KUKA KRL program: MyProgram_094().src

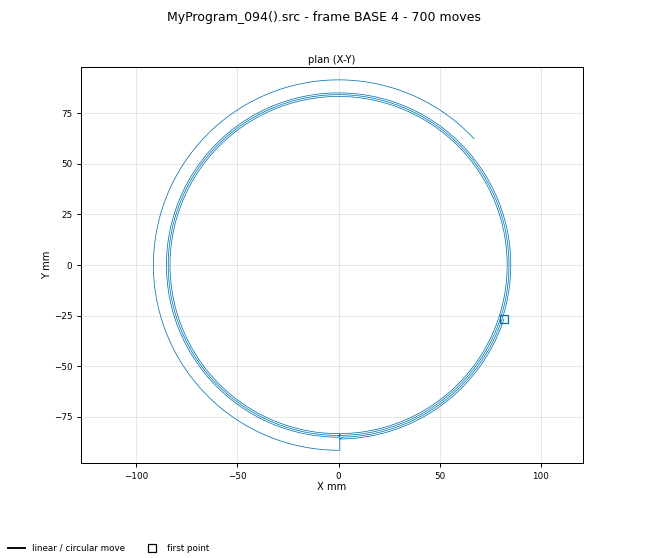
[picture p0: tool path of MyProgram_094().src in frame BASE 4, 700 of 700 moves have a stored position in this frame; points joined in program order, loops and branches not executed]
&ACCESS RVP
&REL 1
&PARAM TEMPLATE = C:\KRC\Roboter\Template\vorgabe
&PARAM EDITMASK = *
DEF MyProgram_094()
; ---- Setting reference (Base) ----
$BASE = BASE_DATA[4]

; --------------------------
; ---- Setting tool (TCP) ----
$TOOL = TOOL_DATA[3]
; --------------------------

$VEL.CP = VEL_APROX_PRINT
Startdeposition()
$VEL.CP = VEL_PRINT
LIN {X 81.733,Y -26.6851,Z 88,A -23.6392,B 24.9182,C -2.0882,E1 25.1514,E2 468.5643} C_DIS
LIN {X 80.2475,Y -30.8683,Z 88,A -26.5648,B 24.9188,C -2.0802,E1 25.1486,E2 471.4924} C_DIS
LIN {X 77.8159,Y -36.5664,Z 88,A -30.6029,B 24.9196,C -2.0708,E1 25.1441,E2 475.5307} C_DIS
LIN {X 76.3718,Y -39.4947,Z 88,A -32.5846,B 24.9196,C -2.071,E1 25.1416,E2 477.5014} C_DIS
LIN {X 74.1282,Y -43.5589,Z 88,A -35.9674,B 24.921,C -2.0522,E1 25.1369,E2 480.911} C_DIS
LIN {X 71.5565,Y -47.6671,Z 88,A -38.965,B 24.9211,C -2.051,E1 25.1324,E2 483.8964} C_DIS
LIN {X 70.1934,Y -49.6508,Z 88,A -41.3471,B 24.9235,C -2.0204,E1 25.1285,E2 486.3392} C_DIS
LIN {X 67.8657,Y -52.7894,Z 88,A -43.5721,B 24.923,C -2.0261,E1 25.1247,E2 488.5401} C_DIS
LIN {X 64.4289,Y -56.934,Z 88,A -46.6091,B 24.9223,C -2.0354,E1 25.1193,E2 491.5414} C_DIS
LIN {X 62.1331,Y -59.4299,Z 88,A -49.1933,B 24.9236,C -2.0188,E1 25.1144,E2 494.1534} C_DIS
LIN {X 59.2198,Y -62.3328,Z 88,A -52.3338,B 24.9251,C -1.999,E1 25.108,E2 497.3276} C_DIS
LIN {X 56.7113,Y -64.6234,Z 88,A -53.6632,B 24.9231,C -2.0249,E1 25.1054,E2 498.5904} C_DIS
LIN {X 54.5742,Y -66.438,Z 88,A -56.1783,B 24.9251,C -1.9992,E1 25.0998,E2 501.1567} C_DIS
LIN {X 49.6783,Y -70.1747,Z 88,A -60.1672,B 24.9254,C -1.9944,E1 25.0909,E2 505.1426} C_DIS
LIN {X 47.2805,Y -71.8114,Z 88,A -62.4831,B 24.9266,C -1.9781,E1 25.0854,E2 507.4893} C_DIS
LIN {X 44.2965,Y -73.6906,Z 88,A -64.087,B 24.9251,C -1.9982,E1 25.0817,E2 509.0406} C_DIS
LIN {X 41.297,Y -75.4121,Z 88,A -66.6065,B 24.926,C -1.9871,E1 25.0756,E2 511.5791} C_DIS
LIN {X 38.2378,Y -77.0077,Z 88,A -68.7734,B 24.926,C -1.9876,E1 25.0702,E2 513.7388} C_DIS
LIN {X 34.3008,Y -78.8402,Z 88,A -72.2408,B 24.9276,C -1.9646,E1 25.0612,E2 517.2521} C_DIS
LIN {X 31.2368,Y -80.1038,Z 88,A -73.7753,B 24.9262,C -1.9833,E1 25.0574,E2 518.7388} C_DIS
LIN {X 28.0288,Y -81.2822,Z 88,A -76.7376,B 24.9281,C -1.9583,E1 25.0494,E2 521.7543} C_DIS
LIN {X 24.8043,Y -82.3237,Z 88,A -78.4493,B 24.927,C -1.9732,E1 25.045,E2 523.4276} C_DIS
LIN {X 21.2594,Y -83.3089,Z 88,A -81.7956,B 24.9293,C -1.9422,E1 25.0358,E2 526.8422} C_DIS
LIN {X 16.7926,Y -84.3241,Z 88,A -83.7415,B 24.9269,C -1.9746,E1 25.0307,E2 528.7088} C_DIS
LIN {X 10.7108,Y -85.3095,Z 88,A -87.865,B 24.9272,C -1.9711,E1 25.0193,E2 532.8369} C_DIS
LIN {X 7.4694,Y -85.6546,Z 88,A -90.1854,B 24.9276,C -1.9652,E1 25.0128,E2 535.1697} C_DIS
LIN {X 4.6796,Y -85.8512,Z 88,A -92.9626,B 24.9297,C -1.9359,E1 25.0049,E2 538.0153} C_DIS
LIN {X 0.5582,Y -85.9679,Z 88,A -93.1523,B 24.9238,C -2.0159,E1 25.0049,E2 538.0153} C_DIS
Enddeposition()
LIN {X 0.5582,Y -85.9679,Z 88,A -93.1523,B 24.9238,C -2.0159,E1 25.0049,E2 538.0153} C_DIS
Startdeposition()
$VEL.CP = VEL_PRINT
LIN {X 1.674,Y -85.0811,Z 88,A -92.9521,B 24.924,C -2.0134,E1 25.0054,E2 537.8212} C_DIS
LIN {X 5.5624,Y -84.9157,Z 88,A -89.8499,B 24.9227,C -2.0298,E1 25.0141,E2 534.6812} C_DIS
LIN {X 9.1586,Y -84.6037,Z 88,A -87.9756,B 24.924,C -2.0134,E1 25.0192,E2 532.8471} C_DIS
LIN {X 12.5486,Y -84.1684,Z 88,A -85.0762,B 24.9224,C -2.0342,E1 25.0274,E2 529.901} C_DIS
LIN {X 16.1894,Y -83.5434,Z 88,A -83.3504,B 24.9241,C -2.0116,E1 25.032,E2 528.2306} C_DIS
LIN {X 20.7796,Y -82.5225,Z 88,A -80.0885,B 24.9237,C -2.0177,E1 25.0409,E2 524.9588} C_DIS
LIN {X 23.9194,Y -81.6672,Z 88,A -77.9107,B 24.9235,C -2.0197,E1 25.0467,E2 522.78} C_DIS
LIN {X 26.4302,Y -80.8894,Z 88,A -75.3855,B 24.9215,C -2.0465,E1 25.0536,E2 520.1959} C_DIS
LIN {X 30.2485,Y -79.5401,Z 88,A -73.5932,B 24.9235,C -2.0195,E1 25.0581,E2 518.4715} C_DIS
LIN {X 33.1948,Y -78.3563,Z 88,A -71.1205,B 24.9225,C -2.0335,E1 25.0645,E2 515.9712} C_DIS
LIN {X 36.3155,Y -76.9608,Z 88,A -68.9238,B 24.9225,C -2.0336,E1 25.0701,E2 513.7799} C_DIS
LIN {X 39.5256,Y -75.3613,Z 88,A -66.5837,B 24.9223,C -2.0352,E1 25.0759,E2 511.4426} C_DIS
LIN {X 42.557,Y -73.692,Z 88,A -64.2486,B 24.922,C -2.0395,E1 25.0816,E2 509.1042} C_DIS
LIN {X 47.2525,Y -70.7745,Z 88,A -60.7688,B 24.922,C -2.0385,E1 25.0898,E2 505.638} C_DIS
LIN {X 50.0783,Y -68.8026,Z 88,A -58.0174,B 24.9206,C -2.0576,E1 25.0961,E2 502.8509} C_DIS
LIN {X 53.2996,Y -66.3382,Z 88,A -55.444,B 24.9206,C -2.0582,E1 25.1017,E2 500.2856} C_DIS
LIN {X 56.1485,Y -63.9452,Z 88,A -52.9116,B 24.9201,C -2.0648,E1 25.1071,E2 497.7476} C_DIS
LIN {X 58.92,Y -61.4008,Z 88,A -50.5533,B 24.9201,C -2.0648,E1 25.1119,E2 495.3988} C_DIS
LIN {X 61.2054,Y -59.1226,Z 88,A -48.345,B 24.9195,C -2.0714,E1 25.1162,E2 493.1845} C_DIS
LIN {X 63.807,Y -56.3066,Z 88,A -45.7587,B 24.919,C -2.078,E1 25.1211,E2 490.594} C_DIS
LIN {X 66.1479,Y -53.5354,Z 88,A -43.3524,B 24.9186,C -2.0832,E1 25.1254,E2 488.1866} C_DIS
LIN {X 68.597,Y -50.3592,Z 88,A -40.3906,B 24.9173,C -2.0994,E1 25.1304,E2 485.2007} C_DIS
LIN {X 70.5872,Y -47.5297,Z 88,A -37.8925,B 24.9164,C -2.1116,E1 25.1343,E2 482.6861} C_DIS
LIN {X 73.7566,Y -42.4447,Z 88,A -34.5122,B 24.9172,C -2.1007,E1 25.1391,E2 479.3487} C_DIS
LIN {X 74.9881,Y -40.2309,Z 88,A -32.7904,B 24.9168,C -2.1062,E1 25.1414,E2 477.623} C_DIS
LIN {X 76.4162,Y -37.4472,Z 88,A -30.7153,B 24.9164,C -2.1114,E1 25.1441,E2 475.5467} C_DIS
LIN {X 77.6659,Y -34.7797,Z 88,A -28.1064,B 24.9142,C -2.1389,E1 25.1471,E2 472.8871} C_DIS
LIN {X 78.9315,Y -31.804,Z 88,A -26.5631,B 24.9154,C -2.1236,E1 25.1487,E2 471.3883} C_DIS
LIN {X 80.7731,Y -26.7857,Z 88,A -22.8946,B 24.9143,C -2.1371,E1 25.1522,E2 467.7086} C_DIS
LIN {X 81.7527,Y -23.6278,Z 88,A -20.5927,B 24.9136,C -2.1466,E1 25.154,E2 465.3972} C_DIS
LIN {X 82.5245,Y -20.7718,Z 88,A -18.9002,B 24.9139,C -2.1426,E1 25.1552,E2 463.724} C_DIS
LIN {X 83.2588,Y -17.6004,Z 88,A -16.4666,B 24.9127,C -2.1579,E1 25.1567,E2 461.2684} C_DIS
LIN {X 84.1496,Y -12.6706,Z 88,A -13.1028,B 24.9118,C -2.1683,E1 25.1583,E2 457.8998} C_DIS
LIN {X 84.5645,Y -9.5168,Z 88,A -11.0727,B 24.9116,C -2.1713,E1 25.1589,E2 455.8746} C_DIS
LIN {X 84.7904,Y -7.2374,Z 88,A -9.3098,B 24.9105,C -2.1839,E1 25.1594,E2 454.0925} C_DIS
LIN {X 85.0939,Y -0.8863,Z 88,A -4.8253,B 24.9088,C -2.2046,E1 25.1598,E2 449.5858} C_DIS
LIN {X 85.0004,Y 4.0858,Z 88,A -1.7552,B 24.9088,C -2.2056,E1 25.1595,E2 446.5315} C_DIS
LIN {X 84.6266,Y 8.9405,Z 88,A 0.8808,B 24.9097,C -2.194,E1 25.1589,E2 443.9385} C_DIS
LIN {X 84.3639,Y 11.1521,Z 88,A 3.4937,B 24.9061,C -2.237,E1 25.1579,E2 441.2396} C_DIS
LIN {X 83.7907,Y 14.8575,Z 88,A 5.1462,B 24.908,C -2.2148,E1 25.1572,E2 439.6491} C_DIS
LIN {X 83.0057,Y 18.7565,Z 88,A 8.0759,B 24.9066,C -2.2317,E1 25.1555,E2 436.6967} C_DIS
LIN {X 82.2132,Y 21.9689,Z 88,A 10.2169,B 24.9063,C -2.2355,E1 25.154,E2 434.559} C_DIS
LIN {X 81.1968,Y 25.4703,Z 88,A 12.5277,B 24.906,C -2.238,E1 25.1521,E2 432.2556} C_DIS
LIN {X 80.3027,Y 28.1614,Z 88,A 14.4713,B 24.9055,C -2.2448,E1 25.1504,E2 430.3068} C_DIS
LIN {X 79.2539,Y 30.9907,Z 88,A 16.5091,B 24.905,C -2.2509,E1 25.1483,E2 428.2659} C_DIS
LIN {X 78.0763,Y 33.8481,Z 88,A 18.5822,B 24.9045,C -2.2566,E1 25.1461,E2 426.1907} C_DIS
LIN {X 76.2957,Y 37.6904,Z 88,A 21.4623,B 24.9037,C -2.2656,E1 25.1426,E2 423.3051} C_DIS
LIN {X 75.2676,Y 39.7036,Z 88,A 23.177,B 24.9028,C -2.2762,E1 25.1404,E2 421.5741} C_DIS
LIN {X 73.4534,Y 42.9689,Z 88,A 25.4627,B 24.9028,C -2.2752,E1 25.1372,E2 419.3027} C_DIS
LIN {X 71.9394,Y 45.4587,Z 88,A 27.564,B 24.902,C -2.285,E1 25.1341,E2 417.1889} C_DIS
LIN {X 69.9909,Y 48.4035,Z 88,A 29.4184,B 24.903,C -2.2735,E1 25.1313,E2 415.3709} C_DIS
LIN {X 68.6867,Y 50.2366,Z 88,A 31.7063,B 24.9005,C -2.3031,E1 25.1274,E2 413.024} C_DIS
LIN {X 65.9916,Y 53.7283,Z 88,A 34.3193,B 24.9009,C -2.2982,E1 25.1229,E2 410.4348} C_DIS
LIN {X 63.8485,Y 56.2591,Z 88,A 36.2398,B 24.9014,C -2.2929,E1 25.1195,E2 408.5355} C_DIS
LIN {X 61.2216,Y 59.1058,Z 88,A 39.0377,B 24.9003,C -2.3049,E1 25.1141,E2 405.7215} C_DIS
LIN {X 58.927,Y 61.394,Z 88,A 41.2254,B 24.8999,C -2.3097,E1 25.1097,E2 403.5316} C_DIS
LIN {X 57.0263,Y 63.1642,Z 88,A 43.4545,B 24.8982,C -2.3291,E1 25.105,E2 401.2657} C_DIS
LIN {X 53.3912,Y 66.2648,Z 88,A 46.3212,B 24.8987,C -2.3236,E1 25.0989,E2 398.423} C_DIS
LIN {X 50.359,Y 68.5971,Z 88,A 48.6255,B 24.8991,C -2.3192,E1 25.0938,E2 396.1373} C_DIS
LIN {X 47.5261,Y 70.5897,Z 88,A 51.2112,B 24.898,C -2.3313,E1 25.0878,E2 393.5317} C_DIS
LIN {X 43.9489,Y 72.8708,Z 88,A 54.1354,B 24.8974,C -2.3378,E1 25.0809,E2 390.6014} C_DIS
LIN {X 40.6311,Y 74.771,Z 88,A 56.4193,B 24.898,C -2.332,E1 25.0754,E2 388.338} C_DIS
LIN {X 37.416,Y 76.4317,Z 88,A 58.942,B 24.8974,C -2.3378,E1 25.0691,E2 385.8084} C_DIS
LIN {X 33.4143,Y 78.2638,Z 88,A 62.1381,B 24.8965,C -2.3486,E1 25.0608,E2 382.5946} C_DIS
LIN {X 29.8776,Y 79.6805,Z 88,A 64.4126,B 24.8971,C -2.3418,E1 25.055,E2 380.3411} C_DIS
LIN {X 26.993,Y 80.7032,Z 88,A 66.5381,B 24.8968,C -2.3456,E1 25.0494,E2 378.2108} C_DIS
LIN {X 24.0987,Y 81.614,Z 88,A 68.2506,B 24.8975,C -2.3368,E1 25.0448,E2 376.5225} C_DIS
LIN {X 22.2097,Y 82.1481,Z 88,A 69.9297,B 24.8965,C -2.3489,E1 25.0403,E2 374.8174} C_DIS
LIN {X 18.6575,Y 83.0286,Z 88,A 72.4715,B 24.8961,C -2.3526,E1 25.0333,E2 372.2702} C_DIS
LIN {X 15.4369,Y 83.6865,Z 88,A 74.8346,B 24.8957,C -2.3582,E1 25.0268,E2 369.8966} C_DIS
LIN {X 11.3965,Y 84.3322,Z 88,A 78.0857,B 24.8942,C -2.3744,E1 25.0177,E2 366.6098} C_DIS
LIN {X 7.2412,Y 84.7901,Z 88,A 79.8785,B 24.897,C -2.343,E1 25.013,E2 364.8928} C_DIS
LIN {X 2.2359,Y 85.0689,Z 88,A 83.2687,B 24.897,C -2.3433,E1 25.0035,E2 361.503} C_DIS
LIN {X -2.7082,Y 85.0544,Z 88,A 86.7497,B 24.8966,C -2.3471,E1 24.9938,E2 358.0127} C_DIS
LIN {X -5.3566,Y 84.9296,Z 88,A 88.6724,B 24.8963,C -2.3506,E1 24.9884,E2 356.0812} C_DIS
LIN {X -9.5041,Y 84.5656,Z 88,A 91.7516,B 24.8957,C -2.3575,E1 24.9798,E2 352.9838} C_DIS
LIN {X -13.7307,Y 83.983,Z 88,A 94.3168,B 24.8967,C -2.3463,E1 24.9728,E2 350.443} C_DIS
LIN {X -16.67,Y 83.45,Z 88,A 96.6213,B 24.8961,C -2.3535,E1 24.9664,E2 348.1189} C_DIS
LIN {X -20.4797,Y 82.597,Z 88,A 99.096,B 24.8967,C -2.3464,E1 24.9597,E2 345.6577} C_DIS
LIN {X -23.8514,Y 81.6874,Z 88,A 101.249,B 24.8974,C -2.3381,E1 24.954,E2 343.5211} C_DIS
LIN {X -26.5654,Y 80.8456,Z 88,A 102.9762,B 24.8981,C -2.3304,E1 24.9494,E2 341.8091} C_DIS
LIN {X -28.6735,Y 80.1229,Z 88,A 105.3821,B 24.8959,C -2.3552,E1 24.9429,E2 339.3393} C_DIS
LIN {X -32.1339,Y 78.7972,Z 88,A 107.0664,B 24.8983,C -2.3279,E1 24.9387,E2 337.7163} C_DIS
LIN {X -34.1412,Y 77.9486,Z 88,A 109.3024,B 24.8965,C -2.3483,E1 24.9329,E2 335.4263} C_DIS
LIN {X -37.4433,Y 76.4182,Z 88,A 111.4142,B 24.8977,C -2.3345,E1 24.9276,E2 333.342} C_DIS
LIN {X -41.7912,Y 74.1296,Z 88,A 114.2929,B 24.8993,C -2.3165,E1 24.9206,E2 330.4981} C_DIS
LIN {X -43.4835,Y 73.1492,Z 88,A 115.6929,B 24.8993,C -2.3165,E1 24.9172,E2 329.0938} C_DIS
LIN {X -46.9211,Y 70.993,Z 88,A 118.4101,B 24.8998,C -2.3109,E1 24.9109,E2 326.3812} C_DIS
LIN {X -49.5289,Y 69.1989,Z 88,A 120.7052,B 24.8998,C -2.3114,E1 24.9056,E2 324.0772} C_DIS
LIN {X -52.2836,Y 67.1431,Z 88,A 123.2689,B 24.8996,C -2.3137,E1 24.8999,E2 321.4987} C_DIS
LIN {X -56.5544,Y 63.5866,Z 88,A 126.7808,B 24.9009,C -2.2988,E1 24.8925,E2 318.0086} C_DIS
LIN {X -59.0838,Y 61.2429,Z 88,A 128.7809,B 24.9021,C -2.2843,E1 24.8885,E2 316.0349} C_DIS
LIN {X -61.8922,Y 58.4035,Z 88,A 132.2962,B 24.9007,C -2.3011,E1 24.8815,E2 312.4643} C_DIS
LIN {X -64.0589,Y 56.0182,Z 88,A 133.956,B 24.9024,C -2.2812,E1 24.8785,E2 310.8446} C_DIS
LIN {X -66.0527,Y 53.6529,Z 88,A 136.1086,B 24.9027,C -2.2778,E1 24.8747,E2 308.6903} C_DIS
LIN {X -68.813,Y 50.0642,Z 88,A 139.321,B 24.903,C -2.2742,E1 24.8693,E2 305.4709} C_DIS
LIN {X -70.7985,Y 47.2161,Z 88,A 141.5882,B 24.9037,C -2.2658,E1 24.8658,E2 303.2125} C_DIS
LIN {X -72.8663,Y 43.9564,Z 88,A 143.8101,B 24.9052,C -2.248,E1 24.8625,E2 301.0217} C_DIS
LIN {X -74.6995,Y 40.7629,Z 88,A 146.5667,B 24.9052,C -2.2485,E1 24.8587,E2 298.2494} C_DIS
LIN {X -76.0148,Y 38.257,Z 88,A 149.7014,B 24.9027,C -2.2774,E1 24.8547,E2 295.029} C_DIS
LIN {X -78.2713,Y 33.3967,Z 88,A 152.1988,B 24.9063,C -2.2354,E1 24.852,E2 292.6181} C_DIS
LIN {X -79.537,Y 30.2567,Z 88,A 154.6707,B 24.9063,C -2.2338,E1 24.8495,E2 290.1361} C_DIS
LIN {X -81.0653,Y 25.8863,Z 88,A 157.2835,B 24.9084,C -2.2102,E1 24.8472,E2 287.5647} C_DIS
LIN {X -82.6653,Y 20.1997,Z 88,A 161.4624,B 24.9089,C -2.2032,E1 24.8441,E2 283.3782} C_DIS
LIN {X -83.2818,Y 17.4863,Z 88,A 164.23,B 24.9074,C -2.2221,E1 24.8425,E2 280.5493} C_DIS
LIN {X -84.0159,Y 13.5278,Z 88,A 166.3708,B 24.9094,C -2.1976,E1 24.8415,E2 278.4542} C_DIS
LIN {X -84.5217,Y 9.8824,Z 88,A 168.6155,B 24.9106,C -2.1833,E1 24.8407,E2 276.2304} C_DIS
LIN {X -84.8054,Y 7.0493,Z 88,A 170.7697,B 24.9106,C -2.1837,E1 24.8402,E2 274.0623} C_DIS
LIN {X -85.0355,Y 3.2706,Z 88,A 173.0826,B 24.9118,C -2.169,E1 24.8399,E2 271.7705} C_DIS
LIN {X -85.0953,Y 0.7104,Z 88,A 175.0169,B 24.9118,C -2.1693,E1 24.8398,E2 269.8238} C_DIS
LIN {X -85.0787,Y -1.8025,Z 88,A 176.7265,B 24.9121,C -2.1644,E1 24.8398,E2 268.1156} C_DIS
LIN {X -84.8988,Y -5.8126,Z 88,A 179.3735,B 24.913,C -2.1543,E1 24.8403,E2 265.4769} C_DIS
LIN {X -84.5915,Y -9.275,Z 88,A -178.4267,B 24.9139,C -2.143,E1 24.8409,E2 263.2908} C_DIS
LIN {X -84.1274,Y -12.8142,Z 88,A -176.2543,B 24.915,C -2.1291,E1 24.8417,E2 261.1386} C_DIS
LIN {X -83.6684,Y -15.5375,Z 88,A -173.9271,B 24.9144,C -2.1362,E1 24.8428,E2 258.7806} C_DIS
LIN {X -83.016,Y -18.7118,Z 88,A -171.7739,B 24.915,C -2.1287,E1 24.8441,E2 256.6327} C_DIS
LIN {X -82.2299,Y -21.9068,Z 88,A -169.5865,B 24.9156,C -2.1212,E1 24.8456,E2 254.4504} C_DIS
LIN {X -81.3524,Y -24.9687,Z 88,A -167.7614,B 24.9168,C -2.1059,E1 24.847,E2 252.6513} C_DIS
LIN {X -80.1201,Y -28.6812,Z 88,A -164.0907,B 24.9151,C -2.1272,E1 24.8504,E2 248.909} C_DIS
LIN {X -78.8162,Y -32.0872,Z 88,A -162.6711,B 24.918,C -2.091,E1 24.8518,E2 247.5678} C_DIS
LIN {X -76.524,Y -37.2267,Z 88,A -158.3562,B 24.9177,C -2.095,E1 24.8569,E2 243.2197} C_DIS
LIN {X -74.9156,Y -40.3646,Z 88,A -156.1092,B 24.9185,C -2.0849,E1 24.8598,E2 240.9847} C_DIS
LIN {X -73.8012,Y -42.367,Z 88,A -153.6123,B 24.9167,C -2.108,E1 24.8634,E2 238.4197} C_DIS
LIN {X -71.4346,Y -46.2471,Z 88,A -151.6177,B 24.9197,C -2.0697,E1 24.8662,E2 236.5065} C_DIS
LIN {X -67.4963,Y -51.8252,Z 88,A -146.8622,B 24.9202,C -2.0628,E1 24.874,E2 231.7443} C_DIS
LIN {X -64.6921,Y -55.2859,Z 88,A -143.8328,B 24.9207,C -2.0567,E1 24.8793,E2 228.7154} C_DIS
LIN {X -62.5161,Y -57.7355,Z 88,A -141.5614,B 24.9209,C -2.0536,E1 24.8836,E2 226.4412} C_DIS
LIN {X -60.1802,Y -60.168,Z 88,A -139.2525,B 24.9212,C -2.0499,E1 24.8881,E2 224.1313} C_DIS
LIN {X -58.3015,Y -61.9881,Z 88,A -137.4532,B 24.9214,C -2.0475,E1 24.8918,E2 222.3304} C_DIS
LIN {X -55.7513,Y -64.292,Z 88,A -135.2197,B 24.9219,C -2.0406,E1 24.8964,E2 220.1044} C_DIS
LIN {X -52.9553,Y -66.6137,Z 88,A -132.2458,B 24.9211,C -2.0516,E1 24.903,E2 217.0932} C_DIS
LIN {X -50.3771,Y -68.5839,Z 88,A -130.6259,B 24.9226,C -2.0312,E1 24.9065,E2 215.5161} C_DIS
LIN {X -46.5617,Y -71.23,Z 88,A -126.9572,B 24.9218,C -2.0422,E1 24.9151,E2 211.8089} C_DIS
LIN {X -42.6057,Y -73.664,Z 88,A -124.2644,B 24.9231,C -2.0248,E1 24.9215,E2 209.1495} C_DIS
LIN {X -39.7318,Y -75.2527,Z 88,A -122.152,B 24.9236,C -2.0189,E1 24.9267,E2 207.045} C_DIS
LIN {X -36.4408,Y -76.9016,Z 88,A -119.6826,B 24.9238,C -2.0156,E1 24.9328,E2 204.5769} C_DIS
LIN {X -34.2773,Y -77.8893,Z 88,A -118.1507,B 24.9241,C -2.0118,E1 24.9367,E2 203.0505} C_DIS
LIN {X -31.1024,Y -79.21,Z 88,A -115.7422,B 24.9241,C -2.0123,E1 24.943,E2 200.6353} C_DIS
LIN {X -28.1418,Y -80.3095,Z 88,A -113.5508,B 24.9241,C -2.0124,E1 24.9487,E2 198.4393} C_DIS
LIN {X -23.3302,Y -81.8371,Z 88,A -110.1376,B 24.9242,C -2.0104,E1 24.9579,E2 195.025} C_DIS
LIN {X -19.7979,Y -82.7634,Z 88,A -107.7916,B 24.9246,C -2.0056,E1 24.9642,E2 192.6872} C_DIS
LIN {X -16.0378,Y -83.5726,Z 88,A -105.0987,B 24.9244,C -2.0077,E1 24.9716,E2 189.9862} C_DIS
LIN {X -12.2846,Y -84.2061,Z 88,A -102.3734,B 24.9241,C -2.012,E1 24.9791,E2 187.2481} C_DIS
LIN {X -5.3558,Y -84.9296,Z 88,A -98.1217,B 24.9252,C -1.9979,E1 24.9909,E2 183.0276} C_DIS
LIN {X -0.18,Y -85.098,Z 88,A -94.2404,B 24.9242,C -2.0108,E1 25.0018,E2 179.1154} C_DIS
LIN {X -0.18,Y -85.098,Z 88,A -94.2404,B 24.9242,C -2.0108,E1 25.0018,E2 179.1154} C_DIS
Enddeposition()
LIN {X 0.5449,Y -84.2116,Z 88,A -94.4053,B 24.9246,C -2.0058,E1 25.0013,E2 179.292} C_DIS
Startdeposition()
$VEL.CP = VEL_PRINT
LIN {X -3.9343,Y -84.1248,Z 88,A -97.867,B 24.9256,C -1.9926,E1 24.9915,E2 182.7855} C_DIS
LIN {X -8.021,Y -83.834,Z 88,A -100.384,B 24.9249,C -2.0009,E1 24.9846,E2 185.2839} C_DIS
LIN {X -12.8471,Y -83.2307,Z 88,A -103.938,B 24.9254,C -1.9941,E1 24.9747,E2 188.8567} C_DIS
LIN {X -15.5725,Y -82.7649,Z 88,A -105.9884,B 24.9258,C -1.9896,E1 24.969,E2 190.9197} C_DIS
LIN {X -18.2227,Y -82.2217,Z 88,A -107.7908,B 24.9256,C -1.9916,E1 24.9641,E2 192.7197} C_DIS
LIN {X -21.4532,Y -81.4397,Z 88,A -109.842,B 24.9251,C -1.9991,E1 24.9586,E2 194.7559} C_DIS
LIN {X -23.603,Y -80.842,Z 88,A -111.5897,B 24.9255,C -1.9933,E1 24.9538,E2 196.5202} C_DIS
LIN {X -26.1064,Y -80.0681,Z 88,A -113.3313,B 24.9253,C -1.9958,E1 24.9492,E2 198.2588} C_DIS
LIN {X -29.3486,Y -78.9387,Z 88,A -115.4867,B 24.9248,C -2.0031,E1 24.9436,E2 200.4012} C_DIS
LIN {X -34.1042,Y -77.003,Z 88,A -118.943,B 24.9244,C -2.0077,E1 24.9347,E2 203.8543} C_DIS
LIN {X -36.3696,Y -75.9583,Z 88,A -120.8192,B 24.9247,C -2.0045,E1 24.9299,E2 205.743} C_DIS
LIN {X -39.0543,Y -74.6137,Z 88,A -122.8892,B 24.9245,C -2.0063,E1 24.9248,E2 207.8144} C_DIS
LIN {X -41.84,Y -73.0879,Z 88,A -125.1197,B 24.9245,C -2.0072,E1 24.9193,E2 210.0492} C_DIS
LIN {X -45.7024,Y -70.7372,Z 88,A -128.6838,B 24.9252,C -1.9979,E1 24.9108,E2 213.6466} C_DIS
LIN {X -48.3682,Y -68.9424,Z 88,A -130.4194,B 24.9239,C -2.0143,E1 24.9069,E2 215.3492} C_DIS
LIN {X -52.3131,Y -65.9982,Z 88,A -133.5009,B 24.9229,C -2.0277,E1 24.9001,E2 218.4097} C_DIS
LIN {X -54.2922,Y -64.3812,Z 88,A -135.5198,B 24.9233,C -2.023,E1 24.8957,E2 220.4475} C_DIS
LIN {X -56.7741,Y -62.2025,Z 88,A -137.6335,B 24.9226,C -2.0312,E1 24.8913,E2 222.5502} C_DIS
LIN {X -58.8916,Y -60.2025,Z 88,A -139.7767,B 24.9226,C -2.0307,E1 24.887,E2 224.7034} C_DIS
LIN {X -61.2663,Y -57.7828,Z 88,A -142.0384,B 24.9222,C -2.0369,E1 24.8826,E2 226.9601} C_DIS
LIN {X -63.5312,Y -55.283,Z 88,A -144.3631,B 24.9219,C -2.0413,E1 24.8783,E2 229.2849} C_DIS
LIN {X -65.6801,Y -52.7132,Z 88,A -146.5372,B 24.9212,C -2.0495,E1 24.8745,E2 231.4495} C_DIS
LIN {X -68.3713,Y -49.1718,Z 88,A -149.3762,B 24.9203,C -2.062,E1 24.8697,E2 234.2723} C_DIS
LIN {X -69.8916,Y -46.9856,Z 88,A -151.5628,B 24.9207,C -2.0562,E1 24.8662,E2 236.4836} C_DIS
LIN {X -71.6656,Y -44.234,Z 88,A -154.0257,B 24.9207,C -2.0555,E1 24.8626,E2 238.9606} C_DIS
LIN {X -73.7184,Y -40.7204,Z 88,A -156.6079,B 24.9198,C -2.0679,E1 24.859,E2 241.5267} C_DIS
LIN {X -75.0516,Y -38.2057,Z 88,A -158.3968,B 24.9191,C -2.0773,E1 24.8567,E2 243.3028} C_DIS
LIN {X -76.815,Y -34.5234,Z 88,A -161.2097,B 24.9185,C -2.0841,E1 24.8534,E2 246.1148} C_DIS
LIN {X -78.0561,Y -31.6176,Z 88,A -163.42,B 24.9182,C -2.0886,E1 24.851,E2 248.3266} C_DIS
LIN {X -79.2769,Y -28.4215,Z 88,A -166.4986,B 24.9192,C -2.0752,E1 24.848,E2 251.4545} C_DIS
LIN {X -80.4734,Y -24.8282,Z 88,A -168.1059,B 24.9166,C -2.1089,E1 24.8468,E2 252.9906} C_DIS
LIN {X -81.0897,Y -22.7358,Z 88,A -169.9518,B 24.917,C -2.1036,E1 24.8453,E2 254.8599} C_DIS
LIN {X -81.9922,Y -19.229,Z 88,A -172.3613,B 24.9163,C -2.1126,E1 24.8437,E2 257.2621} C_DIS
LIN {X -82.5668,Y -16.5905,Z 88,A -174.3043,B 24.9161,C -2.1154,E1 24.8426,E2 259.2098} C_DIS
LIN {X -83.1963,Y -13.0695,Z 88,A -176.6715,B 24.9153,C -2.1247,E1 24.8415,E2 261.5688} C_DIS
LIN {X -83.6519,Y -9.7349,Z 88,A -178.9276,B 24.9147,C -2.1328,E1 24.8407,E2 263.819} C_DIS
LIN {X -83.9623,Y -6.5392,Z 88,A 178.8783,B 24.9142,C -2.1395,E1 24.8402,E2 266.0105} C_DIS
LIN {X -84.1273,Y -3.8827,Z 88,A 176.9926,B 24.9138,C -2.1432,E1 24.8399,E2 267.8986} C_DIS
LIN {X -84.2153,Y -0.4717,Z 88,A 174.6826,B 24.9132,C -2.1509,E1 24.8398,E2 270.2041} C_DIS
LIN {X -84.1686,Y 2.8503,Z 88,A 172.377,B 24.9127,C -2.1569,E1 24.8399,E2 272.5092} C_DIS
LIN {X -83.9935,Y 6.1399,Z 88,A 170.0903,B 24.9123,C -2.1629,E1 24.8403,E2 274.7954} C_DIS
LIN {X -83.675,Y 9.5377,Z 88,A 167.7854,B 24.9116,C -2.1708,E1 24.841,E2 277.0953} C_DIS
LIN {X -83.3008,Y 12.388,Z 88,A 165.3564,B 24.9121,C -2.1644,E1 24.842,E2 279.5539} C_DIS
LIN {X -82.133,Y 18.6196,Z 88,A 161.7101,B 24.9096,C -2.1958,E1 24.844,E2 283.1468} C_DIS
LIN {X -80.9632,Y 23.1821,Z 88,A 158.4783,B 24.9088,C -2.2052,E1 24.8463,E2 286.3751} C_DIS
LIN {X -80.2983,Y 25.3929,Z 88,A 156.2644,B 24.9098,C -2.1929,E1 24.8481,E2 288.631} C_DIS
LIN {X -78.9485,Y 29.3219,Z 88,A 153.8831,B 24.9081,C -2.2134,E1 24.8503,E2 290.9769} C_DIS
LIN {X -77.9739,Y 31.8194,Z 88,A 152.1217,B 24.9075,C -2.2206,E1 24.8521,E2 292.7308} C_DIS
LIN {X -76.9486,Y 34.2268,Z 88,A 150.308,B 24.9071,C -2.2251,E1 24.8542,E2 294.544} C_DIS
LIN {X -75.2282,Y 37.8601,Z 88,A 147.391,B 24.9069,C -2.2283,E1 24.8577,E2 297.4692} C_DIS
LIN {X -74.0041,Y 40.1969,Z 88,A 145.5673,B 24.9065,C -2.2327,E1 24.8601,E2 299.2918} C_DIS
LIN {X -72.6885,Y 42.5314,Z 88,A 143.7868,B 24.9059,C -2.2391,E1 24.8626,E2 301.0665} C_DIS
LIN {X -70.9616,Y 45.3528,Z 88,A 141.5664,B 24.9053,C -2.2462,E1 24.8659,E2 303.2811} C_DIS
LIN {X -69.1811,Y 48.0247,Z 88,A 139.4777,B 24.9046,C -2.2548,E1 24.8691,E2 305.3597} C_DIS
LIN {X -67.4676,Y 50.4041,Z 88,A 137.7165,B 24.9036,C -2.2666,E1 24.872,E2 307.1014} C_DIS
LIN {X -65.9576,Y 52.3644,Z 88,A 135.7186,B 24.904,C -2.2625,E1 24.8755,E2 309.1186} C_DIS
LIN {X -64.0644,Y 54.6641,Z 88,A 133.698,B 24.9035,C -2.2678,E1 24.8791,E2 311.1357} C_DIS
LIN {X -61.8188,Y 57.1922,Z 88,A 131.2398,B 24.9034,C -2.2693,E1 24.8837,E2 313.6014} C_DIS
LIN {X -60.1758,Y 58.9187,Z 88,A 129.6261,B 24.903,C -2.2734,E1 24.8868,E2 315.2121} C_DIS
LIN {X -57.9264,Y 61.1313,Z 88,A 127.5389,B 24.9025,C -2.2801,E1 24.891,E2 317.2921} C_DIS
LIN {X -55.4982,Y 63.3432,Z 88,A 125.2213,B 24.9022,C -2.2829,E1 24.8958,E2 319.6121} C_DIS
LIN {X -53.25,Y 65.2451,Z 88,A 123.3815,B 24.9015,C -2.2918,E1 24.8997,E2 321.4377} C_DIS
LIN {X -51.1064,Y 66.9378,Z 88,A 121.3624,B 24.9015,C -2.2913,E1 24.9042,E2 323.4656} C_DIS
LIN {X -48.5201,Y 68.8363,Z 88,A 119.1443,B 24.9012,C -2.2947,E1 24.9093,E2 325.6832} C_DIS
LIN {X -45.8613,Y 70.6352,Z 88,A 116.8956,B 24.901,C -2.2971,E1 24.9145,E2 327.9336} C_DIS
LIN {X -42.8432,Y 72.5042,Z 88,A 114.6647,B 24.9002,C -2.3067,E1 24.9198,E2 330.1486} C_DIS
LIN {X -40.3323,Y 73.9307,Z 88,A 111.991,B 24.9016,C -2.2902,E1 24.9264,E2 332.8691} C_DIS
LIN {X -37.2059,Y 75.5524,Z 88,A 109.8762,B 24.9006,C -2.3019,E1 24.9317,E2 334.9617} C_DIS
LIN {X -33.5727,Y 77.2352,Z 88,A 107.4466,B 24.8995,C -2.3143,E1 24.9378,E2 337.3678} C_DIS
LIN {X -28.3744,Y 79.2941,Z 88,A 103.5898,B 24.8992,C -2.3178,E1 24.9479,E2 341.2244} C_DIS
LIN {X -25.191,Y 80.3609,Z 88,A 101.3393,B 24.8989,C -2.3214,E1 24.9538,E2 343.4702} C_DIS
LIN {X -22.0268,Y 81.2848,Z 88,A 99.2373,B 24.8983,C -2.3278,E1 24.9594,E2 345.5603} C_DIS
LIN {X -19.2311,Y 81.9917,Z 88,A 97.2131,B 24.8983,C -2.3278,E1 24.9649,E2 347.5872} C_DIS
LIN {X -16.3858,Y 82.6083,Z 88,A 95.1124,B 24.8985,C -2.3261,E1 24.9707,E2 349.6947} C_DIS
LIN {X -13.1808,Y 83.1791,Z 88,A 93.05,B 24.898,C -2.3321,E1 24.9763,E2 351.7448} C_DIS
LIN {X -10.3531,Y 83.5782,Z 88,A 90.7866,B 24.8987,C -2.3239,E1 24.9827,E2 354.0292} C_DIS
LIN {X -6.3152,Y 83.9802,Z 88,A 88.3302,B 24.8978,C -2.3342,E1 24.9894,E2 356.4626} C_DIS
LIN {X -3.6993,Y 84.1351,Z 88,A 86.5717,B 24.8977,C -2.3355,E1 24.9943,E2 358.2183} C_DIS
LIN {X -0.2807,Y 84.2162,Z 88,A 83.7299,B 24.8989,C -2.3209,E1 25.0024,E2 361.095} C_DIS
LIN {X 3.0882,Y 84.1612,Z 88,A 81.7155,B 24.8982,C -2.3293,E1 25.0079,E2 363.089} C_DIS
LIN {X 6.5858,Y 83.9586,Z 88,A 79.5201,B 24.8977,C -2.3349,E1 25.014,E2 365.2702} C_DIS
LIN {X 10.3006,Y 83.5856,Z 88,A 77.0869,B 24.8975,C -2.3377,E1 25.0207,E2 367.6951} C_DIS
LIN {X 12.508,Y 83.2831,Z 88,A 75.3207,B 24.8982,C -2.3298,E1 25.0257,E2 369.4785} C_DIS
LIN {X 15.168,Y 82.8396,Z 88,A 73.5249,B 24.8982,C -2.3303,E1 25.0306,E2 371.2712} C_DIS
LIN {X 18.4584,Y 82.1702,Z 88,A 71.4581,B 24.8976,C -2.3358,E1 25.0362,E2 373.3222} C_DIS
LIN {X 20.6573,Y 81.6442,Z 88,A 69.7064,B 24.8983,C -2.3284,E1 25.041,E2 375.0888} C_DIS
LIN {X 24.0215,Y 80.7178,Z 88,A 67.318,B 24.8985,C -2.3263,E1 25.0474,E2 377.4781} C_DIS
LIN {X 27.4109,Y 79.6322,Z 88,A 65.1394,B 24.898,C -2.3318,E1 25.0531,E2 379.6395} C_DIS
LIN {X 29.9331,Y 78.7173,Z 88,A 63.1162,B 24.8987,C -2.324,E1 25.0585,E2 381.677} C_DIS
LIN {X 32.4817,Y 77.7007,Z 88,A 61.2847,B 24.8987,C -2.3232,E1 25.0632,E2 383.5062} C_DIS
LIN {X 35.0696,Y 76.5689,Z 88,A 59.1793,B 24.8994,C -2.3153,E1 25.0686,E2 385.6251} C_DIS
LIN {X 38.4062,Y 74.9491,Z 88,A 56.7925,B 24.8994,C -2.3164,E1 25.0745,E2 388.0028} C_DIS
LIN {X 41.4949,Y 73.2859,Z 88,A 54.0731,B 24.9005,C -2.3027,E1 25.0812,E2 390.7467} C_DIS
LIN {X 46.1743,Y 70.43,Z 88,A 51.0064,B 24.8992,C -2.3179,E1 25.0884,E2 393.7676} C_DIS
LIN {X 48.2776,Y 69.0053,Z 88,A 49.2415,B 24.8995,C -2.3139,E1 25.0925,E2 395.536} C_DIS
LIN {X 50.2436,Y 67.5882,Z 88,A 47.4616,B 24.9002,C -2.3069,E1 25.0965,E2 397.3262} C_DIS
LIN {X 52.3814,Y 65.9442,Z 88,A 45.5119,B 24.9008,C -2.2999,E1 25.1008,E2 399.2852} C_DIS
LIN {X 55.4637,Y 63.3734,Z 88,A 42.8944,B 24.9008,C -2.2983,E1 25.1064,E2 401.8963} C_DIS
LIN {X 57.7266,Y 61.3191,Z 88,A 40.8075,B 24.9013,C -2.2939,E1 25.1106,E2 403.9852} C_DIS
LIN {X 60.2391,Y 58.8546,Z 88,A 38.3446,B 24.9019,C -2.2866,E1 25.1155,E2 406.4549} C_DIS
LIN {X 62.5864,Y 56.3507,Z 88,A 36.3433,B 24.9014,C -2.2923,E1 25.1193,E2 408.4341} C_DIS
LIN {X 64.0585,Y 54.6709,Z 88,A 34.546,B 24.9025,C -2.2798,E1 25.1226,E2 410.2527} C_DIS
LIN {X 66.147,Y 52.1247,Z 88,A 31.5459,B 24.905,C -2.25,E1 25.1279,E2 413.3093} C_DIS
LIN {X 68.5486,Y 48.9234,Z 88,A 29.9152,B 24.9026,C -2.2787,E1 25.1305,E2 414.8643} C_DIS
LIN {X 69.9496,Y 46.8999,Z 88,A 27.8642,B 24.904,C -2.2621,E1 25.1337,E2 416.9443} C_DIS
LIN {X 71.8272,Y 43.9696,Z 88,A 25.5532,B 24.9044,C -2.2578,E1 25.1372,E2 419.2537} C_DIS
LIN {X 73.2024,Y 41.6407,Z 88,A 23.6281,B 24.905,C -2.2501,E1 25.1399,E2 421.1871} C_DIS
LIN {X 74.6259,Y 39.0311,Z 88,A 21.6923,B 24.9052,C -2.2474,E1 25.1424,E2 423.119} C_DIS
LIN {X 76.1211,Y 36.0305,Z 88,A 19.3364,B 24.906,C -2.2386,E1 25.1453,E2 425.4832} C_DIS
LIN {X 77.6493,Y 32.6038,Z 88,A 16.8857,B 24.9063,C -2.2347,E1 25.148,E2 427.9296} C_DIS
LIN {X 78.9513,Y 29.3142,Z 88,A 14.456,B 24.907,C -2.2269,E1 25.1504,E2 430.3642} C_DIS
LIN {X 80.1161,Y 25.958,Z 88,A 12.1516,B 24.9073,C -2.2235,E1 25.1525,E2 432.6636} C_DIS
LIN {X 81.0705,Y 22.8037,Z 88,A 9.9076,B 24.9078,C -2.2167,E1 25.1542,E2 434.9109} C_DIS
LIN {X 81.902,Y 19.6109,Z 88,A 7.6524,B 24.9084,C -2.2095,E1 25.1558,E2 437.1701} C_DIS
LIN {X 82.5744,Y 16.5536,Z 88,A 5.4535,B 24.9092,C -2.2006,E1 25.157,E2 439.3771} C_DIS
LIN {X 83.5565,Y 10.5264,Z 88,A 2.0414,B 24.9082,C -2.2125,E1 25.1585,E2 442.7411} C_DIS
LIN {X 84.0609,Y 5.1252,Z 88,A -2.5225,B 24.9115,C -2.1716,E1 25.1596,E2 447.3746} C_DIS
LIN {X 84.2119,Y 0.9937,Z 88,A -5.0123,B 24.9115,C -2.1733,E1 25.1598,E2 449.8454} C_DIS
LIN {X 84.1981,Y -1.7709,Z 88,A -7.0937,B 24.9124,C -2.1606,E1 25.1597,E2 451.9445} C_DIS
LIN {X 84.0557,Y -5.2204,Z 88,A -9.205,B 24.9124,C -2.161,E1 25.1594,E2 454.0422} C_DIS
LIN {X 83.8264,Y -8.1037,Z 88,A -11.1572,B 24.9129,C -2.1553,E1 25.1589,E2 455.9965} C_DIS
LIN {X 83.483,Y -11.0935,Z 88,A -13.1718,B 24.9133,C -2.1498,E1 25.1582,E2 458.012} C_DIS
LIN {X 83.0926,Y -13.7134,Z 88,A -15.0998,B 24.9141,C -2.1399,E1 25.1574,E2 459.9523} C_DIS
LIN {X 82.6048,Y -16.4041,Z 88,A -16.6934,B 24.9139,C -2.1429,E1 25.1565,E2 461.5294} C_DIS
LIN {X 81.9918,Y -19.2308,Z 88,A -18.7682,B 24.9147,C -2.133,E1 25.1553,E2 463.6154} C_DIS
LIN {X 81.1899,Y -22.3783,Z 88,A -20.9977,B 24.9153,C -2.1254,E1 25.1537,E2 465.85} C_DIS
LIN {X 80.2681,Y -25.4881,Z 88,A -23.2174,B 24.9159,C -2.1181,E1 25.1518,E2 468.0744} C_DIS
LIN {X 79.3274,Y -28.2797,Z 88,A -25.3312,B 24.9166,C -2.1082,E1 25.1499,E2 470.1995} C_DIS
LIN {X 78.3014,Y -31.0055,Z 88,A -27.2907,B 24.9171,C -2.1029,E1 25.1479,E2 472.1608} C_DIS
LIN {X 76.9007,Y -34.3332,Z 88,A -29.5859,B 24.9172,C -2.1009,E1 25.1454,E2 474.4483} C_DIS
LIN {X 75.5179,Y -37.2756,Z 88,A -31.7535,B 24.9176,C -2.0958,E1 25.1427,E2 476.6163} C_DIS
LIN {X 73.9996,Y -40.2052,Z 88,A -33.8844,B 24.9178,C -2.093,E1 25.14,E2 478.7425} C_DIS
LIN {X 71.6738,Y -44.2209,Z 88,A -37.2293,B 24.919,C -2.0777,E1 25.1352,E2 482.1064} C_DIS
LIN {X 69.8556,Y -47.0387,Z 88,A -39.3974,B 24.9193,C -2.0751,E1 25.1319,E2 484.2698} C_DIS
LIN {X 66.7356,Y -51.3689,Z 88,A -42.8376,B 24.9195,C -2.0715,E1 25.1262,E2 487.7017} C_DIS
LIN {X 63.5217,Y -55.2939,Z 88,A -46.3528,B 24.9204,C -2.0604,E1 25.1199,E2 491.227} C_DIS
LIN {X 60.9108,Y -58.1571,Z 88,A -49.2041,B 24.9214,C -2.0468,E1 25.1145,E2 494.0981} C_DIS
LIN {X 57.9459,Y -61.1115,Z 88,A -52.1918,B 24.9223,C -2.0354,E1 25.1084,E2 497.1003} C_DIS
LIN {X 55.0386,Y -63.7447,Z 88,A -55.5751,B 24.9245,C -2.0062,E1 25.1012,E2 500.5392} C_DIS
LIN {X 51.3576,Y -66.7443,Z 88,A -57.6776,B 24.9223,C -2.0357,E1 25.0967,E2 502.5642} C_DIS
LIN {X 49.0348,Y -68.469,Z 88,A -59.7065,B 24.9228,C -2.0296,E1 25.0921,E2 504.6002} C_DIS
LIN {X 46.3166,Y -70.3362,Z 88,A -62.2086,B 24.9237,C -2.0169,E1 25.0863,E2 507.1242} C_DIS
LIN {X 43.5467,Y -72.0842,Z 88,A -64.1739,B 24.9234,C -2.0211,E1 25.0817,E2 509.0731} C_DIS
LIN {X 40.8211,Y -73.6622,Z 88,A -66.3384,B 24.9237,C -2.0166,E1 25.0764,E2 511.2418} C_DIS
LIN {X 37.9601,Y -75.1771,Z 88,A -68.5614,B 24.9241,C -2.0123,E1 25.0709,E2 513.469} C_DIS
LIN {X 35.0599,Y -76.5732,Z 88,A -70.7492,B 24.9243,C -2.0089,E1 25.0653,E2 515.6592} C_DIS
LIN {X 32.0791,Y -77.8682,Z 88,A -72.9616,B 24.9246,C -2.0057,E1 25.0596,E2 517.874} C_DIS
LIN {X 28.1465,Y -79.3741,Z 88,A -75.4347,B 24.9239,C -2.0143,E1 25.0532,E2 520.3215} C_DIS
LIN {X 26.0201,Y -80.096,Z 88,A -77.2448,B 24.9247,C -2.0034,E1 25.0484,E2 522.1537} C_DIS
LIN {X 23.097,Y -80.9873,Z 88,A -79.3447,B 24.925,C -2.0005,E1 25.0428,E2 524.257} C_DIS
LIN {X 20.184,Y -81.7622,Z 88,A -81.4733,B 24.9253,C -1.9959,E1 25.037,E2 526.3932} C_DIS
LIN {X 17.6972,Y -82.3364,Z 88,A -83.1063,B 24.9252,C -1.9976,E1 25.0325,E2 528.0201} C_DIS
LIN {X 14.3419,Y -82.9875,Z 88,A -85.4364,B 24.9253,C -1.9955,E1 25.0261,E2 530.3525} C_DIS
LIN {X 11.568,Y -83.4186,Z 88,A -87.3194,B 24.9253,C -1.995,E1 25.0209,E2 532.2348} C_DIS
LIN {X 8.6656,Y -83.7694,Z 88,A -89.4289,B 24.9257,C -1.9902,E1 25.015,E2 534.3544} C_DIS
LIN {X 3.0239,Y -84.1632,Z 88,A -92.9736,B 24.9252,C -1.9978,E1 25.0052,E2 537.8795} C_DIS
LIN {X 0.5449,Y -84.2116,Z 88,A -94.4041,B 24.9246,C -2.0053,E1 25.0013,E2 539.292} C_DIS
Enddeposition()
LIN {X 0.5449,Y -84.2116,Z 88,A -94.4041,B 24.9246,C -2.0053,E1 25.0013,E2 539.292} C_DIS
Startdeposition()
$VEL.CP = VEL_PRINT
LIN {X 1.0163,Y -83.3306,Z 88,A -93.759,B 24.9227,C -2.0305,E1 25.0033,E2 538.5873} C_DIS
LIN {X 3.0486,Y -83.281,Z 88,A -92.3623,B 24.9227,C -2.0309,E1 25.0071,E2 537.1899} C_DIS
LIN {X 5.0772,Y -83.1819,Z 88,A -90.9673,B 24.9227,C -2.0314,E1 25.011,E2 535.7942} C_DIS
LIN {X 7.0991,Y -83.0336,Z 88,A -89.5705,B 24.9226,C -2.0322,E1 25.0149,E2 534.3963} C_DIS
LIN {X 9.1934,Y -82.8282,Z 88,A -88.1347,B 24.9226,C -2.0327,E1 25.0189,E2 532.9602} C_DIS
LIN {X 11.2172,Y -82.5785,Z 88,A -86.7308,B 24.9225,C -2.0336,E1 25.0228,E2 531.5553} C_DIS
LIN {X 13.6633,Y -82.2076,Z 88,A -84.8951,B 24.922,C -2.0391,E1 25.0279,E2 529.7084} C_DIS
LIN {X 16.8713,Y -81.6097,Z 88,A -82.7211,B 24.922,C -2.0388,E1 25.0339,E2 527.5376} C_DIS
LIN {X 20.2582,Y -80.8371,Z 88,A -80.414,B 24.922,C -2.0385,E1 25.0401,E2 525.2345} C_DIS
LIN {X 22.2313,Y -80.3169,Z 88,A -78.9516,B 24.9218,C -2.0419,E1 25.0441,E2 523.7665} C_DIS
LIN {X 24.191,Y -79.7485,Z 88,A -77.609,B 24.9218,C -2.0416,E1 25.0477,E2 522.4269} C_DIS
LIN {X 26.1297,Y -79.1344,Z 88,A -76.2146,B 24.9218,C -2.0431,E1 25.0514,E2 521.0315} C_DIS
LIN {X 28.6803,Y -78.2447,Z 88,A -74.1172,B 24.9209,C -2.0532,E1 25.0569,E2 518.9145} C_DIS
LIN {X 31.9059,Y -76.9872,Z 88,A -71.9913,B 24.9213,C -2.0484,E1 25.0624,E2 516.8048} C_DIS
LIN {X 33.7871,Y -76.1803,Z 88,A -70.5881,B 24.9212,C -2.0503,E1 25.066,E2 515.4004} C_DIS
LIN {X 35.6362,Y -75.3332,Z 88,A -69.1946,B 24.921,C -2.0524,E1 25.0695,E2 514.0056} C_DIS
LIN {X 37.4702,Y -74.438,Z 88,A -67.5531,B 24.9202,C -2.0623,E1 25.0737,E2 512.345} C_DIS
LIN {X 40.1786,Y -73.0117,Z 88,A -65.6984,B 24.9206,C -2.0579,E1 25.0782,E2 510.5061} C_DIS
LIN {X 41.9542,Y -72.006,Z 88,A -64.3008,B 24.9204,C -2.0602,E1 25.0816,E2 509.1072} C_DIS
LIN {X 43.7044,Y -70.9573,Z 88,A -62.6934,B 24.9197,C -2.0695,E1 25.0855,E2 507.4829} C_DIS
LIN {X 46.3065,Y -69.2873,Z 88,A -60.7809,B 24.9199,C -2.0667,E1 25.0899,E2 505.5834} C_DIS
LIN {X 47.9838,Y -68.1365,Z 88,A -59.395,B 24.9197,C -2.0691,E1 25.0931,E2 504.1965} C_DIS
LIN {X 49.6318,Y -66.9455,Z 88,A -57.7913,B 24.919,C -2.0787,E1 25.0967,E2 502.5758} C_DIS
LIN {X 52.0425,Y -65.0889,Z 88,A -55.7157,B 24.9187,C -2.0827,E1 25.1013,E2 500.4985} C_DIS
LIN {X 54.4449,Y -63.0933,Z 88,A -53.5794,B 24.9183,C -2.0871,E1 25.1058,E2 498.3599} C_DIS
LIN {X 56.6773,Y -61.0955,Z 88,A -51.5457,B 24.918,C -2.0911,E1 25.11,E2 496.3251} C_DIS
LIN {X 58.7816,Y -59.0727,Z 88,A -49.5388,B 24.9176,C -2.0959,E1 25.114,E2 494.3152} C_DIS
LIN {X 61.0902,Y -56.6831,Z 88,A -47.2716,B 24.9172,C -2.101,E1 25.1184,E2 492.0459} C_DIS
LIN {X 63.091,Y -54.4476,Z 88,A -45.2093,B 24.9168,C -2.1062,E1 25.1222,E2 489.9805} C_DIS
LIN {X 65.0026,Y -52.1499,Z 88,A -43.1966,B 24.9165,C -2.1102,E1 25.1257,E2 487.9677} C_DIS
LIN {X 67.1031,Y -49.4166,Z 88,A -41.1849,B 24.9169,C -2.1047,E1 25.1291,E2 485.9785} C_DIS
LIN {X 68.4906,Y -47.4744,Z 88,A -39.3112,B 24.916,C -2.1169,E1 25.1321,E2 484.0852} C_DIS
LIN {X 70.0727,Y -45.1065,Z 88,A -37.2917,B 24.9154,C -2.1244,E1 25.1352,E2 482.0579} C_DIS
LIN {X 71.4709,Y -42.8594,Z 88,A -35.6307,B 24.9154,C -2.1244,E1 25.1377,E2 480.4057} C_DIS
LIN {X 72.4943,Y -41.1045,Z 88,A -34.239,B 24.9151,C -2.1282,E1 25.1396,E2 479.0121} C_DIS
LIN {X 73.5009,Y -39.2765,Z 88,A -32.8183,B 24.9148,C -2.1319,E1 25.1415,E2 477.5901} C_DIS
LIN {X 74.4407,Y -37.4647,Z 88,A -31.424,B 24.9145,C -2.1357,E1 25.1433,E2 476.1941} C_DIS
LIN {X 75.333,Y -35.6366,Z 88,A -30.0332,B 24.9141,C -2.1396,E1 25.1449,E2 474.8015} C_DIS
LIN {X 76.1858,Y -33.7751,Z 88,A -28.6348,B 24.9138,C -2.1436,E1 25.1465,E2 473.4016} C_DIS
LIN {X 77.0216,Y -31.8218,Z 88,A -27.1503,B 24.9134,C -2.1488,E1 25.1482,E2 471.9129} C_DIS
LIN {X 78.1232,Y -29.0133,Z 88,A -25.125,B 24.913,C -2.1535,E1 25.1502,E2 469.8877} C_DIS
LIN {X 78.81,Y -27.0923,Z 88,A -23.7321,B 24.9127,C -2.1575,E1 25.1515,E2 468.4932} C_DIS
LIN {X 79.4478,Y -25.161,Z 88,A -22.2599,B 24.9121,C -2.1643,E1 25.1527,E2 467.0132} C_DIS
LIN {X 80.0401,Y -23.208,Z 88,A -20.9454,B 24.9121,C -2.1658,E1 25.1538,E2 465.7028} C_DIS
LIN {X 80.5844,Y -21.241,Z 88,A -19.4793,B 24.9115,C -2.1723,E1 25.1548,E2 464.2297} C_DIS
LIN {X 81.0804,Y -19.2613,Z 88,A -17.9226,B 24.9107,C -2.1819,E1 25.1559,E2 462.6594} C_DIS
LIN {X 81.7369,Y -16.2514,Z 88,A -15.8519,B 24.9103,C -2.187,E1 25.157,E2 460.5887} C_DIS
LIN {X 82.2809,Y -13.224,Z 88,A -13.9639,B 24.9103,C -2.1861,E1 25.1579,E2 458.7138} C_DIS
LIN {X 82.5799,Y -11.2065,Z 88,A -12.4293,B 24.9096,C -2.1951,E1 25.1585,E2 457.1671} C_DIS
LIN {X 82.9356,Y -8.1678,Z 88,A -10.477,B 24.9095,C -2.1967,E1 25.1591,E2 455.2225} C_DIS
LIN {X 83.1106,Y -6.136,Z 88,A -9.0843,B 24.9091,C -2.2009,E1 25.1594,E2 453.8282} C_DIS
LIN {X 83.2358,Y -4.101,Z 88,A -7.5077,B 24.9083,C -2.2113,E1 25.1597,E2 452.2365} C_DIS
LIN {X 83.3307,Y -1.0108,Z 88,A -5.5623,B 24.9083,C -2.212,E1 25.1597,E2 450.3009} C_DIS
LIN {X 83.3307,Y 1.0125,Z 88,A -4.1998,B 24.9079,C -2.2155,E1 25.1597,E2 448.9383} C_DIS
LIN {X 83.2811,Y 3.0456,Z 88,A -2.8119,B 24.9076,C -2.2196,E1 25.1597,E2 447.549} C_DIS
LIN {X 83.182,Y 5.0749,Z 88,A -1.4253,B 24.9072,C -2.2237,E1 25.1594,E2 446.1609} C_DIS
LIN {X 83.0284,Y 7.1625,Z 88,A 0.2318,B 24.9062,C -2.2356,E1 25.159,E2 444.4856} C_DIS
LIN {X 82.7112,Y 10.192,Z 88,A 2.0839,B 24.9064,C -2.2341,E1 25.1585,E2 442.648} C_DIS
LIN {X 82.4384,Y 12.2035,Z 88,A 3.4698,B 24.906,C -2.2381,E1 25.1579,E2 441.2607} C_DIS
LIN {X 82.0681,Y 14.4798,Z 88,A 4.8942,B 24.906,C -2.2377,E1 25.1573,E2 439.8458} C_DIS
LIN {X 81.7367,Y 16.2526,Z 88,A 6.2973,B 24.9053,C -2.247,E1 25.1565,E2 438.4289} C_DIS
LIN {X 81.3096,Y 18.2694,Z 88,A 7.6785,B 24.905,C -2.2501,E1 25.1557,E2 437.0483} C_DIS
LIN {X 80.8378,Y 20.2552,Z 88,A 9.0738,B 24.9047,C -2.2541,E1 25.1548,E2 435.6516} C_DIS
LIN {X 80.0411,Y 23.2043,Z 88,A 11.1641,B 24.9042,C -2.2601,E1 25.1532,E2 433.559} C_DIS
LIN {X 79.4438,Y 25.1736,Z 88,A 12.5688,B 24.9038,C -2.264,E1 25.152,E2 432.1532} C_DIS
LIN {X 78.8031,Y 27.1128,Z 88,A 13.9637,B 24.9035,C -2.2679,E1 25.1508,E2 430.757} C_DIS
LIN {X 78.1126,Y 29.0421,Z 88,A 15.3638,B 24.9032,C -2.2717,E1 25.1494,E2 429.3557} C_DIS
LIN {X 77.38,Y 30.9413,Z 88,A 16.7553,B 24.9029,C -2.2755,E1 25.148,E2 427.963} C_DIS
LIN {X 76.3414,Y 33.4181,Z 88,A 18.6695,B 24.9022,C -2.2831,E1 25.1459,E2 426.0414} C_DIS
LIN {X 75.3313,Y 35.6401,Z 88,A 20.2557,B 24.9021,C -2.2847,E1 25.1441,E2 424.4599} C_DIS
LIN {X 74.4372,Y 37.4717,Z 88,A 21.8663,B 24.9011,C -2.2955,E1 25.142,E2 422.8324} C_DIS
LIN {X 73.007,Y 40.1871,Z 88,A 23.7474,B 24.9013,C -2.2937,E1 25.1396,E2 420.9655} C_DIS
LIN {X 72.0004,Y 41.9639,Z 88,A 25.1436,B 24.901,C -2.2972,E1 25.1376,E2 419.5683} C_DIS
LIN {X 70.9506,Y 43.7155,Z 88,A 26.5417,B 24.9007,C -2.3007,E1 25.1356,E2 418.1691} C_DIS
LIN {X 69.8581,Y 45.4408,Z 88,A 27.9361,B 24.9004,C -2.304,E1 25.1335,E2 416.7738} C_DIS
LIN {X 68.3381,Y 47.6938,Z 88,A 29.8413,B 24.8999,C -2.3099,E1 25.1305,E2 414.864} C_DIS
LIN {X 66.5429,Y 50.1681,Z 88,A 32.1696,B 24.8988,C -2.3225,E1 25.1266,E2 412.5172} C_DIS
LIN {X 64.4211,Y 52.8673,Z 88,A 34.4506,B 24.8985,C -2.3254,E1 25.1226,E2 410.2398} C_DIS
LIN {X 62.4289,Y 55.2056,Z 88,A 36.5531,B 24.8981,C -2.3299,E1 25.1187,E2 408.1362} C_DIS
LIN {X 60.3515,Y 57.4692,Z 88,A 38.6502,B 24.8978,C -2.334,E1 25.1147,E2 406.0385} C_DIS
LIN {X 58.1985,Y 59.6487,Z 88,A 40.749,B 24.8974,C -2.3382,E1 25.1106,E2 403.9386} C_DIS
LIN {X 55.9693,Y 61.7451,Z 88,A 42.8426,B 24.8971,C -2.3421,E1 25.1063,E2 401.8442} C_DIS
LIN {X 53.6651,Y 63.7579,Z 88,A 44.9398,B 24.8967,C -2.346,E1 25.1018,E2 399.7461} C_DIS
LIN {X 51.2686,Y 65.7005,Z 88,A 46.8336,B 24.897,C -2.3426,E1 25.0977,E2 397.8675} C_DIS
LIN {X 49.6445,Y 66.9362,Z 88,A 48.2327,B 24.8968,C -2.3449,E1 25.0946,E2 396.4679} C_DIS
LIN {X 47.9851,Y 68.1356,Z 88,A 49.8173,B 24.8961,C -2.3529,E1 25.0909,E2 394.8699} C_DIS
LIN {X 45.4777,Y 69.8339,Z 88,A 51.709,B 24.8964,C -2.3502,E1 25.0866,E2 392.9908} C_DIS
LIN {X 43.8287,Y 70.8799,Z 88,A 53.3142,B 24.8954,C -2.3606,E1 25.0827,E2 391.3662} C_DIS
LIN {X 41.0706,Y 72.5137,Z 88,A 55.2406,B 24.8959,C -2.355,E1 25.0781,E2 389.4589} C_DIS
LIN {X 39.2815,Y 73.4983,Z 88,A 56.6439,B 24.8958,C -2.3568,E1 25.0747,E2 388.0552} C_DIS
LIN {X 37.3067,Y 74.519,Z 88,A 58.058,B 24.8959,C -2.3552,E1 25.0712,E2 386.6489} C_DIS
LIN {X 35.6345,Y 75.334,Z 88,A 59.4448,B 24.8955,C -2.3601,E1 25.0677,E2 385.2541} C_DIS
LIN {X 33.7751,Y 76.1858,Z 88,A 61.0989,B 24.8946,C -2.3695,E1 25.0634,E2 383.5819} C_DIS
LIN {X 30.9392,Y 77.3808,Z 88,A 62.9575,B 24.8952,C -2.3636,E1 25.0586,E2 381.7415} C_DIS
LIN {X 29.0273,Y 78.1181,Z 88,A 64.3633,B 24.8951,C -2.3649,E1 25.055,E2 380.3357} C_DIS
LIN {X 27.1042,Y 78.806,Z 88,A 65.7648,B 24.895,C -2.366,E1 25.0513,E2 378.9344} C_DIS
LIN {X 25.1712,Y 79.4446,Z 88,A 67.3077,B 24.8945,C -2.3715,E1 25.0471,E2 377.3812} C_DIS
LIN {X 22.2278,Y 80.3178,Z 88,A 69.4285,B 24.8943,C -2.3733,E1 25.0414,E2 375.2598} C_DIS
LIN {X 19.2538,Y 81.0822,Z 88,A 71.3778,B 24.8946,C -2.3696,E1 25.0362,E2 373.3222} C_DIS
LIN {X 17.2554,Y 81.5308,Z 88,A 72.7845,B 24.8946,C -2.3702,E1 25.0324,E2 371.9158} C_DIS
LIN {X 15.0735,Y 81.9614,Z 88,A 74.196,B 24.8948,C -2.3673,E1 25.0285,E2 370.513} C_DIS
LIN {X 13.2307,Y 82.2798,Z 88,A 75.5932,B 24.8945,C -2.3711,E1 25.0246,E2 369.1082} C_DIS
LIN {X 11.2133,Y 82.579,Z 88,A 76.9983,B 24.8945,C -2.3715,E1 25.0208,E2 367.7033} C_DIS
LIN {X 8.6517,Y 82.885,Z 88,A 78.8737,B 24.8942,C -2.3749,E1 25.0155,E2 365.8212} C_DIS
LIN {X 6.128,Y 83.1112,Z 88,A 80.5133,B 24.8944,C -2.3719,E1 25.011,E2 364.1895} C_DIS
LIN {X 4.0965,Y 83.2361,Z 88,A 81.9142,B 24.8944,C -2.3719,E1 25.0071,E2 362.7891} C_DIS
LIN {X 2.0636,Y 83.3112,Z 88,A 83.313,B 24.8944,C -2.3719,E1 25.0032,E2 361.3909} C_DIS
LIN {X 0.0316,Y 83.3367,Z 88,A 84.7104,B 24.8944,C -2.3716,E1 24.9993,E2 359.9942} C_DIS
LIN {X -2.2619,Y 83.3051,Z 88,A 86.1497,B 24.8949,C -2.3671,E1 24.9953,E2 358.5654} C_DIS
LIN {X -4.0914,Y 83.2364,Z 88,A 87.7965,B 24.8939,C -2.3781,E1 24.9906,E2 356.892} C_DIS
LIN {X -7.1342,Y 83.0308,Z 88,A 89.6471,B 24.8946,C -2.37,E1 24.9855,E2 355.06} C_DIS
LIN {X -9.1676,Y 82.831,Z 88,A 91.0536,B 24.8946,C -2.3693,E1 24.9816,E2 353.6543} C_DIS
LIN {X -11.7726,Y 82.4996,Z 88,A 92.956,B 24.8946,C -2.371,E1 24.9763,E2 351.7464} C_DIS
LIN {X -14.2498,Y 82.1095,Z 88,A 94.5869,B 24.8949,C -2.367,E1 24.9719,E2 350.1234} C_DIS
LIN {X -16.2496,Y 81.7372,Z 88,A 95.9897,B 24.8949,C -2.3661,E1 24.968,E2 348.7214} C_DIS
LIN {X -18.6844,Y 81.2137,Z 88,A 97.844,B 24.8947,C -2.3687,E1 24.9629,E2 346.8585} C_DIS
LIN {X -21.4368,Y 80.5315,Z 88,A 99.535,B 24.8956,C -2.3593,E1 24.9584,E2 345.1873} C_DIS
LIN {X -23.2117,Y 80.039,Z 88,A 100.9316,B 24.8953,C -2.3617,E1 24.9547,E2 343.7828} C_DIS
LIN {X -25.1657,Y 79.4463,Z 88,A 102.5934,B 24.8948,C -2.3675,E1 24.9502,E2 342.1042} C_DIS
LIN {X -28.15,Y 78.4381,Z 88,A 104.4811,B 24.8958,C -2.3569,E1 24.9453,E2 340.2382} C_DIS
LIN {X -30.0189,Y 77.7423,Z 88,A 105.8735,B 24.8958,C -2.3557,E1 24.9416,E2 338.8458} C_DIS
LIN {X -32.293,Y 76.8241,Z 88,A 107.7117,B 24.8957,C -2.3577,E1 24.9369,E2 336.9986} C_DIS
LIN {X -34.6945,Y 75.7714,Z 88,A 109.3988,B 24.8962,C -2.3517,E1 24.9326,E2 335.3217} C_DIS
LIN {X -36.5222,Y 74.9075,Z 88,A 110.7774,B 24.8964,C -2.3492,E1 24.9291,E2 333.9455} C_DIS
LIN {X -38.33,Y 73.9986,Z 88,A 112.174,B 24.8966,C -2.3471,E1 24.9256,E2 332.5501} C_DIS
LIN {X -40.1142,Y 73.0466,Z 88,A 113.7506,B 24.8964,C -2.35,E1 24.9218,E2 330.9621} C_DIS
LIN {X -42.8391,Y 71.4831,Z 88,A 115.9918,B 24.8965,C -2.3485,E1 24.9164,E2 328.7179} C_DIS
LIN {X -45.4517,Y 69.851,Z 88,A 117.868,B 24.8975,C -2.3377,E1 24.912,E2 326.8613} C_DIS
LIN {X -47.1484,Y 68.7172,Z 88,A 119.2771,B 24.8977,C -2.3351,E1 24.9087,E2 325.4536} C_DIS
LIN {X -48.8223,Y 67.5382,Z 88,A 120.6868,B 24.8979,C -2.3324,E1 24.9055,E2 324.0457} C_DIS
LIN {X -50.8639,Y 66.0124,Z 88,A 122.5599,B 24.8979,C -2.3321,E1 24.9013,E2 322.1664} C_DIS
LIN {X -53.2516,Y 64.1017,Z 88,A 124.6799,B 24.8983,C -2.328,E1 24.8968,E2 320.0481} C_DIS
LIN {X -55.5859,Y 62.0885,Z 88,A 126.8023,B 24.8987,C -2.3233,E1 24.8923,E2 317.9285} C_DIS
LIN {X -57.8279,Y 60.0058,Z 88,A 128.9188,B 24.8991,C -2.3188,E1 24.888,E2 315.8142} C_DIS
LIN {X -59.9939,Y 57.8403,Z 88,A 131.0357,B 24.8995,C -2.314,E1 24.8839,E2 313.6997} C_DIS
LIN {X -62.0924,Y 55.5815,Z 88,A 133.1643,B 24.9,C -2.309,E1 24.8799,E2 311.5737} C_DIS
LIN {X -64.0916,Y 53.2639,Z 88,A 135.3191,B 24.9003,C -2.3049,E1 24.876,E2 309.4186} C_DIS
LIN {X -66.0061,Y 50.872,Z 88,A 137.4008,B 24.9009,C -2.2987,E1 24.8724,E2 307.3419} C_DIS
LIN {X -67.5286,Y 48.8354,Z 88,A 139.1474,B 24.9013,C -2.294,E1 24.8695,E2 305.5983} C_DIS
LIN {X -68.72,Y 47.1444,Z 88,A 140.4833,B 24.9018,C -2.2877,E1 24.8674,E2 304.2706} C_DIS
LIN {X -69.8541,Y 45.447,Z 88,A 141.8947,B 24.9021,C -2.284,E1 24.8652,E2 302.8609} C_DIS
LIN {X -70.9498,Y 43.7168,Z 88,A 143.3088,B 24.9025,C -2.2802,E1 24.8632,E2 301.4487} C_DIS
LIN {X -71.9991,Y 41.9661,Z 88,A 144.722,B 24.9028,C -2.2765,E1 24.8611,E2 300.0371} C_DIS
LIN {X -73.3011,Y 39.645,Z 88,A 146.6447,B 24.903,C -2.2738,E1 24.8585,E2 298.1108} C_DIS
LIN {X -74.4547,Y 37.4365,Z 88,A 148.2845,B 24.9036,C -2.2667,E1 24.8565,E2 296.479} C_DIS
LIN {X -75.3442,Y 35.6128,Z 88,A 149.6895,B 24.9039,C -2.2629,E1 24.8548,E2 295.0756} C_DIS
LIN {X -76.1949,Y 33.7544,Z 88,A 151.332,B 24.9037,C -2.2651,E1 24.8529,E2 293.4189} C_DIS
LIN {X -77.3791,Y 30.9437,Z 88,A 153.2275,B 24.9047,C -2.2533,E1 24.8509,E2 291.5409} C_DIS
LIN {X -78.1149,Y 29.036,Z 88,A 154.633,B 24.9051,C -2.249,E1 24.8495,E2 290.1377} C_DIS
LIN {X -78.8014,Y 27.1176,Z 88,A 156.2297,B 24.9051,C -2.2499,E1 24.848,E2 288.5297} C_DIS
LIN {X -79.7483,Y 24.1917,Z 88,A 158.1729,B 24.906,C -2.2388,E1 24.8464,E2 286.602} C_DIS
LIN {X -80.3137,Y 22.2423,Z 88,A 159.5776,B 24.9063,C -2.2347,E1 24.8453,E2 285.199} C_DIS
LIN {X -80.9529,Y 19.7838,Z 88,A 161.5097,B 24.9063,C -2.2342,E1 24.844,E2 283.2568} C_DIS
LIN {X -81.5209,Y 17.3013,Z 88,A 163.0992,B 24.9072,C -2.2243,E1 24.8431,E2 281.6815} C_DIS
LIN {X -81.9067,Y 15.3696,Z 88,A 164.4595,B 24.9075,C -2.2202,E1 24.8424,E2 280.323} C_DIS
LIN {X -82.3559,Y 12.7389,Z 88,A 166.4283,B 24.9077,C -2.2179,E1 24.8415,E2 278.3479} C_DIS
LIN {X -82.7162,Y 10.1498,Z 88,A 168.0913,B 24.9085,C -2.2086,E1 24.8409,E2 276.6972} C_DIS
LIN {X -82.9358,Y 8.1659,Z 88,A 169.6492,B 24.9085,C -2.2092,E1 24.8404,E2 275.1286} C_DIS
LIN {X -83.1804,Y 5.1036,Z 88,A 171.6344,B 24.9093,C -2.199,E1 24.84,E2 273.1558} C_DIS
LIN {X -83.2805,Y 3.0649,Z 88,A 173.0479,B 24.9096,C -2.1948,E1 24.8399,E2 271.7438} C_DIS
LIN {X -83.3329,Y 0.7296,Z 88,A 174.8724,B 24.9096,C -2.1956,E1 24.8398,E2 269.9065} C_DIS
LIN {X -83.3118,Y -2.044,Z 88,A 176.5832,B 24.9105,C -2.1842,E1 24.8398,E2 268.2125} C_DIS
LIN {X -83.2321,Y -4.1684,Z 88,A 178.0078,B 24.911,C -2.1786,E1 24.84,E2 266.7928} C_DIS
LIN {X -83.1102,Y -6.1408,Z 88,A 179.4175,B 24.9112,C -2.1756,E1 24.8403,E2 265.3815} C_DIS
LIN {X -82.9357,Y -8.1672,Z 88,A -179.1662,B 24.9115,C -2.1717,E1 24.8407,E2 263.9662} C_DIS
LIN {X -82.7108,Y -10.1955,Z 88,A -177.7556,B 24.9119,C -2.1675,E1 24.8411,E2 262.5572} C_DIS
LIN {X -82.334,Y -12.8804,Z 88,A -175.8095,B 24.9122,C -2.1639,E1 24.8419,E2 260.6081} C_DIS
LIN {X -81.9281,Y -15.2584,Z 88,A -174.2092,B 24.9127,C -2.1572,E1 24.8427,E2 259.0144} C_DIS
LIN {X -81.5281,Y -17.2683,Z 88,A -172.7908,B 24.9131,C -2.1531,E1 24.8435,E2 257.5974} C_DIS
LIN {X -81.082,Y -19.2546,Z 88,A -171.3776,B 24.9134,C -2.1492,E1 24.8444,E2 256.1852} C_DIS
LIN {X -80.5857,Y -21.236,Z 88,A -169.7155,B 24.9131,C -2.1519,E1 24.8456,E2 254.507} C_DIS
LIN {X -79.7326,Y -24.2425,Z 88,A -167.8125,B 24.9142,C -2.1388,E1 24.847,E2 252.6242} C_DIS
LIN {X -79.1206,Y -26.1711,Z 88,A -166.407,B 24.9145,C -2.135,E1 24.8483,E2 251.2196} C_DIS
LIN {X -78.4587,Y -28.0936,Z 88,A -164.9955,B 24.9148,C -2.1313,E1 24.8496,E2 249.809} C_DIS
LIN {X -77.747,Y -30.007,Z 88,A -163.5909,B 24.9151,C -2.1272,E1 24.8509,E2 248.4061} C_DIS
LIN {X -76.9655,Y -31.9575,Z 88,A -162.1756,B 24.9155,C -2.1223,E1 24.8524,E2 246.9948} C_DIS
LIN {X -76.1892,Y -33.7673,Z 88,A -160.7666,B 24.9157,C -2.12,E1 24.854,E2 245.5837} C_DIS
LIN {X -75.3449,Y -35.6111,Z 88,A -159.3634,B 24.916,C -2.1163,E1 24.8557,E2 244.1815} C_DIS
LIN {X -74.4367,Y -37.4727,Z 88,A -157.9042,B 24.9162,C -2.1133,E1 24.8575,E2 242.7216} C_DIS
LIN {X -73.492,Y -39.293,Z 88,A -156.5185,B 24.9166,C -2.1088,E1 24.8593,E2 241.3392} C_DIS
LIN {X -72.5104,Y -41.0765,Z 88,A -154.9589,B 24.9166,C -2.1095,E1 24.8614,E2 239.7699} C_DIS
LIN {X -70.9437,Y -43.7266,Z 88,A -152.9741,B 24.9173,C -2.1003,E1 24.8643,E2 237.7967} C_DIS
LIN {X -69.8544,Y -45.4466,Z 88,A -151.5661,B 24.9175,C -2.0969,E1 24.8664,E2 236.3897} C_DIS
LIN {X -68.7232,Y -47.1396,Z 88,A -150.1597,B 24.9178,C -2.0936,E1 24.8686,E2 234.9842} C_DIS
LIN {X -67.5475,Y -48.8093,Z 88,A -148.4841,B 24.9175,C -2.0977,E1 24.8713,E2 233.2908} C_DIS
LIN {X -65.4447,Y -51.5923,Z 88,A -146.1788,B 24.9181,C -2.0894,E1 24.8753,E2 230.9943} C_DIS
LIN {X -63.428,Y -54.0524,Z 88,A -144.0278,B 24.9186,C -2.0833,E1 24.8791,E2 228.8478} C_DIS
LIN {X -61.4011,Y -56.3443,Z 88,A -141.876,B 24.9189,C -2.08,E1 24.8831,E2 226.6944} C_DIS
LIN {X -59.2889,Y -58.5628,Z 88,A -139.797,B 24.9193,C -2.0747,E1 24.8872,E2 224.619} C_DIS
LIN {X -57.0967,Y -60.702,Z 88,A -137.6795,B 24.9196,C -2.0707,E1 24.8914,E2 222.5022} C_DIS
LIN {X -54.7127,Y -62.8595,Z 88,A -135.5045,B 24.92,C -2.0654,E1 24.896,E2 220.3313} C_DIS
LIN {X -52.4707,Y -64.7425,Z 88,A -133.4268,B 24.9202,C -2.0635,E1 24.9004,E2 218.2502} C_DIS
LIN {X -50.4476,Y -66.3329,Z 88,A -131.5362,B 24.9202,C -2.0638,E1 24.9046,E2 216.352} C_DIS
LIN {X -47.987,Y -68.1343,Z 88,A -129.6698,B 24.9209,C -2.0537,E1 24.9088,E2 214.5032} C_DIS
LIN {X -46.315,Y -69.2815,Z 88,A -128.2709,B 24.9211,C -2.0516,E1 24.9121,E2 213.1046} C_DIS
LIN {X -44.6185,Y -70.386,Z 88,A -126.8744,B 24.9212,C -2.0496,E1 24.9153,E2 211.7083} C_DIS
LIN {X -42.8388,Y -71.4833,Z 88,A -125.433,B 24.9214,C -2.0476,E1 24.9188,E2 210.2672} C_DIS
LIN {X -41.066,Y -72.5162,Z 88,A -124.0231,B 24.9215,C -2.0456,E1 24.9222,E2 208.8578} C_DIS
LIN {X -39.279,Y -73.4995,Z 88,A -122.6122,B 24.9217,C -2.044,E1 24.9257,E2 207.4468} C_DIS
LIN {X -37.4686,Y -74.4388,Z 88,A -121.2045,B 24.9217,C -2.0424,E1 24.9292,E2 206.0391} C_DIS
LIN {X -35.5559,Y -75.3706,Z 88,A -119.7042,B 24.9218,C -2.0418,E1 24.9329,E2 204.5365} C_DIS
LIN {X -32.9729,Y -76.5355,Z 88,A -117.7972,B 24.9221,C -2.0385,E1 24.9378,E2 202.6328} C_DIS
LIN {X -30.9419,Y -77.3798,Z 88,A -116.27,B 24.9221,C -2.0374,E1 24.9418,E2 201.1046} C_DIS
LIN {X -29.0299,Y -78.1172,Z 88,A -114.8579,B 24.9223,C -2.0362,E1 24.9454,E2 199.6925} C_DIS
LIN {X -26.9425,Y -78.8605,Z 88,A -113.4442,B 24.9226,C -2.0317,E1 24.9491,E2 198.2868} C_DIS
LIN {X -25.1751,Y -79.4433,Z 88,A -111.8897,B 24.9221,C -2.0389,E1 24.9533,E2 196.7125} C_DIS
LIN {X -22.2184,Y -80.3204,Z 88,A -109.9313,B 24.9225,C -2.0326,E1 24.9586,E2 194.7656} C_DIS
LIN {X -20.2445,Y -80.8405,Z 88,A -108.5237,B 24.9225,C -2.032,E1 24.9624,E2 193.3576} C_DIS
LIN {X -18.2651,Y -81.3106,Z 88,A -107.12,B 24.9226,C -2.0314,E1 24.9662,E2 191.9534} C_DIS
LIN {X -15.6504,Y -81.8526,Z 88,A -105.2099,B 24.9226,C -2.0329,E1 24.9714,E2 190.0375} C_DIS
LIN {X -13.2405,Y -82.2783,Z 88,A -103.5988,B 24.9227,C -2.0302,E1 24.9759,E2 188.4313} C_DIS
LIN {X -11.148,Y -82.5875,Z 88,A -102.0114,B 24.9224,C -2.034,E1 24.9803,E2 186.8337} C_DIS
LIN {X -8.1752,Y -82.9349,Z 88,A -100.0854,B 24.9228,C -2.0297,E1 24.9856,E2 184.9166} C_DIS
LIN {X -6.1538,Y -83.1092,Z 88,A -98.6904,B 24.9228,C -2.0297,E1 24.9895,E2 183.5211} C_DIS
LIN {X -4.1326,Y -83.2341,Z 88,A -97.2988,B 24.9228,C -2.0297,E1 24.9934,E2 182.1289} C_DIS
LIN {X -2.1087,Y -83.3098,Z 88,A -95.6713,B 24.9222,C -2.0371,E1 24.998,E2 180.4837} C_DIS
LIN {X 0.5429,Y -83.3317,Z 88,A -94.6412,B 24.924,C -2.0133,E1 25.0007,E2 179.51} C_DIS
Enddeposition()
LIN {X 0.6147,Y -91.5303,Z 89,A -94.1305,B 24.9329,C -1.8925,E1 25.0013,E2 179.2861} C_DIS
Startdeposition()
$VEL.CP = VEL_PRINT
LIN {X -2.0415,Y -91.5103,Z 89,A -96.1054,B 24.9336,C -1.8816,E1 24.9957,E2 181.2868} C_DIS
LIN {X -4.4914,Y -91.4238,Z 89,A -97.6211,B 24.9336,C -1.8821,E1 24.9915,E2 182.8017} C_DIS
LIN {X -6.5516,Y -91.2984,Z 89,A -98.9108,B 24.9336,C -1.8821,E1 24.9879,E2 184.0918} C_DIS
LIN {X -8.9719,Y -91.0933,Z 89,A -100.4338,B 24.9336,C -1.8821,E1 24.9837,E2 185.6155} C_DIS
LIN {X -11.2047,Y -90.8457,Z 89,A -101.8404,B 24.9336,C -1.8823,E1 24.9797,E2 187.0226} C_DIS
LIN {X -13.4308,Y -90.5434,Z 89,A -103.3481,B 24.9338,C -1.8793,E1 24.9756,E2 188.5388} C_DIS
LIN {X -16.3049,Y -90.0685,Z 89,A -105.1486,B 24.9337,C -1.8806,E1 24.9706,E2 190.3379} C_DIS
LIN {X -19.5713,Y -89.4156,Z 89,A -107.2184,B 24.9337,C -1.882,E1 24.965,E2 192.4067} C_DIS
LIN {X -22.241,Y -88.7909,Z 89,A -108.8775,B 24.9334,C -1.8848,E1 24.9605,E2 194.0616} C_DIS
LIN {X -24.2155,Y -88.2718,Z 89,A -110.146,B 24.9334,C -1.8859,E1 24.957,E2 195.3294} C_DIS
LIN {X -26.5709,Y -87.5927,Z 89,A -111.6942,B 24.9333,C -1.8865,E1 24.9529,E2 196.8787} C_DIS
LIN {X -28.5176,Y -86.9773,Z 89,A -112.974,B 24.9333,C -1.8874,E1 24.9495,E2 198.1587} C_DIS
LIN {X -30.6435,Y -86.2512,Z 89,A -114.4013,B 24.9332,C -1.8879,E1 24.9457,E2 199.5875} C_DIS
LIN {X -33.3937,Y -85.2235,Z 89,A -116.3282,B 24.9332,C -1.8867,E1 24.9407,E2 201.5213} C_DIS
LIN {X -36.0637,Y -84.1302,Z 89,A -118.0346,B 24.9329,C -1.8918,E1 24.9363,E2 203.2196} C_DIS
LIN {X -37.9307,Y -83.3041,Z 89,A -119.3156,B 24.9329,C -1.8931,E1 24.933,E2 204.5006} C_DIS
LIN {X -40.1483,Y -82.2593,Z 89,A -120.8541,B 24.9327,C -1.8947,E1 24.9292,E2 206.039} C_DIS
LIN {X -42.155,Y -81.2493,Z 89,A -122.2647,B 24.9326,C -1.8964,E1 24.9257,E2 207.4496} C_DIS
LIN {X -44.1362,Y -80.1903,Z 89,A -123.8805,B 24.9329,C -1.8916,E1 24.9216,E2 209.0814} C_DIS
LIN {X -47.0579,Y -78.5114,Z 89,A -125.7907,B 24.9323,C -1.9009,E1 24.9171,E2 210.9752} C_DIS
LIN {X -48.9705,Y -77.3329,Z 89,A -127.2017,B 24.9321,C -1.9028,E1 24.9137,E2 212.386} C_DIS
LIN {X -50.8536,Y -76.1078,Z 89,A -128.6125,B 24.932,C -1.9049,E1 24.9105,E2 213.7965} C_DIS
LIN {X -52.5378,Y -74.9539,Z 89,A -129.9138,B 24.9319,C -1.9063,E1 24.9075,E2 215.099} C_DIS
LIN {X -54.5268,Y -73.5209,Z 89,A -131.4357,B 24.9317,C -1.9093,E1 24.904,E2 216.6191} C_DIS
LIN {X -56.1523,Y -72.2857,Z 89,A -132.737,B 24.9316,C -1.9108,E1 24.9012,E2 217.9214} C_DIS
LIN {X -58.0686,Y -70.7568,Z 89,A -134.2592,B 24.9313,C -1.914,E1 24.8979,E2 219.4418} C_DIS
LIN {X -59.7876,Y -69.3104,Z 89,A -135.6716,B 24.9311,C -1.9165,E1 24.8948,E2 220.8537} C_DIS
LIN {X -61.4695,Y -67.8232,Z 89,A -137.083,B 24.931,C -1.9191,E1 24.8919,E2 222.2647} C_DIS
LIN {X -62.9672,Y -66.4337,Z 89,A -138.3859,B 24.9308,C -1.9209,E1 24.8893,E2 223.5684} C_DIS
LIN {X -64.5786,Y -64.8684,Z 89,A -139.7986,B 24.9306,C -1.9236,E1 24.8864,E2 224.9806} C_DIS
LIN {X -66.143,Y -63.2724,Z 89,A -141.4026,B 24.9309,C -1.9203,E1 24.8833,E2 226.5994} C_DIS
LIN {X -68.4348,Y -60.7863,Z 89,A -143.3128,B 24.9301,C -1.9314,E1 24.8798,E2 228.4918} C_DIS
LIN {X -69.906,Y -59.0885,Z 89,A -144.7263,B 24.9299,C -1.9344,E1 24.8772,E2 229.9045} C_DIS
LIN {X -71.2506,Y -57.4593,Z 89,A -146.0766,B 24.9297,C -1.9366,E1 24.8748,E2 231.2558} C_DIS
LIN {X -72.8462,Y -55.4249,Z 89,A -147.6823,B 24.9294,C -1.9408,E1 24.8721,E2 232.859} C_DIS
LIN {X -74.0634,Y -53.7858,Z 89,A -149.0869,B 24.9294,C -1.9401,E1 24.8697,E2 234.2721} C_DIS
LIN {X -75.8863,Y -51.1808,Z 89,A -151.0021,B 24.9289,C -1.9474,E1 24.8667,E2 236.1794} C_DIS
LIN {X -77.2222,Y -49.143,Z 89,A -152.5027,B 24.9286,C -1.9521,E1 24.8644,E2 237.6765} C_DIS
LIN {X -78.405,Y -47.2331,Z 89,A -153.9168,B 24.9283,C -1.9555,E1 24.8624,E2 239.0897} C_DIS
LIN {X -79.5405,Y -45.2947,Z 89,A -155.2953,B 24.928,C -1.9601,E1 24.8605,E2 240.4644} C_DIS
LIN {X -80.6281,Y -43.329,Z 89,A -156.7645,B 24.9278,C -1.962,E1 24.8585,E2 241.9368} C_DIS
LIN {X -81.6672,Y -41.3373,Z 89,A -158.1611,B 24.9275,C -1.9661,E1 24.8567,E2 243.331} C_DIS
LIN {X -82.6571,Y -39.3206,Z 89,A -159.5944,B 24.9273,C -1.9692,E1 24.855,E2 244.7647} C_DIS
LIN {X -83.6584,Y -37.1444,Z 89,A -161.0864,B 24.927,C -1.9737,E1 24.8533,E2 246.2543} C_DIS
LIN {X -84.4869,Y -35.2174,Z 89,A -162.4246,B 24.9267,C -1.9767,E1 24.8518,E2 247.5927} C_DIS
LIN {X -85.3257,Y -33.1334,Z 89,A -163.8215,B 24.9264,C -1.981,E1 24.8504,E2 248.987} C_DIS
LIN {X -86.1834,Y -30.8369,Z 89,A -165.5668,B 24.9266,C -1.9792,E1 24.8487,E2 250.7467} C_DIS
LIN {X -87.26,Y -27.6438,Z 89,A -167.4891,B 24.9257,C -1.991,E1 24.847,E2 252.6516} C_DIS
LIN {X -87.8538,Y -25.6905,Z 89,A -168.7941,B 24.9254,C -1.9941,E1 24.846,E2 253.9568} C_DIS
LIN {X -88.5113,Y -23.3289,Z 89,A -170.3205,B 24.9251,C -1.999,E1 24.8449,E2 255.4805} C_DIS
LIN {X -89.0572,Y -21.1497,Z 89,A -171.9744,B 24.9253,C -1.9959,E1 24.8438,E2 257.1515} C_DIS
LIN {X -89.7753,Y -17.8574,Z 89,A -173.8601,B 24.9243,C -2.009,E1 24.8427,E2 259.0169} C_DIS
LIN {X -90.1865,Y -15.6488,Z 89,A -175.2759,B 24.924,C -2.0131,E1 24.842,E2 260.4313} C_DIS
LIN {X -90.5434,Y -13.4308,Z 89,A -176.6917,B 24.9237,C -2.0172,E1 24.8414,E2 261.8457} C_DIS
LIN {X -90.9525,Y -10.2926,Z 89,A -178.7053,B 24.9233,C -2.0225,E1 24.8407,E2 263.8587} C_DIS
LIN {X -91.1777,Y -8.0575,Z 89,A 179.8966,B 24.9229,C -2.0272,E1 24.8403,E2 265.254} C_DIS
LIN {X -91.348,Y -5.8174,Z 89,A 178.4624,B 24.9227,C -2.0308,E1 24.84,E2 266.6881} C_DIS
LIN {X -91.4633,Y -3.5739,Z 89,A 177.0649,B 24.9223,C -2.0356,E1 24.8399,E2 268.0828} C_DIS
LIN {X -91.5272,Y -1.1233,Z 89,A 175.2852,B 24.9225,C -2.0332,E1 24.8398,E2 269.8789} C_DIS
LIN {X -91.5103,Y 2.0414,Z 89,A 173.5058,B 24.9215,C -2.0455,E1 24.8398,E2 271.6397} C_DIS
LIN {X -91.3731,Y 5.4083,Z 89,A 171.3813,B 24.9211,C -2.0518,E1 24.8401,E2 273.7618} C_DIS
LIN {X -91.2129,Y 7.6491,Z 89,A 169.9651,B 24.9207,C -2.056,E1 24.8404,E2 275.1765} C_DIS
LIN {X -90.999,Y 9.8731,Z 89,A 168.5547,B 24.9204,C -2.0602,E1 24.8408,E2 276.5856} C_DIS
LIN {X -90.7277,Y 12.1155,Z 89,A 167.1327,B 24.9201,C -2.0644,E1 24.8413,E2 278.0058} C_DIS
LIN {X -90.2845,Y 15.0628,Z 89,A 165.183,B 24.9198,C -2.0679,E1 24.8422,E2 279.9588} C_DIS
LIN {X -89.814,Y 17.6562,Z 89,A 163.6107,B 24.9192,C -2.0755,E1 24.843,E2 281.5224} C_DIS
LIN {X -89.31,Y 20.0552,Z 89,A 162.0657,B 24.9189,C -2.08,E1 24.8439,E2 283.0658} C_DIS
LIN {X -88.8395,Y 22.0419,Z 89,A 160.7787,B 24.9186,C -2.0838,E1 24.8447,E2 284.3512} C_DIS
LIN {X -88.2847,Y 24.1676,Z 89,A 159.3875,B 24.9183,C -2.0876,E1 24.8457,E2 285.7413} C_DIS
LIN {X -87.5927,Y 26.5709,Z 89,A 157.8174,B 24.9179,C -2.0923,E1 24.847,E2 287.3092} C_DIS
LIN {X -86.9142,Y 28.7126,Z 89,A 156.4014,B 24.9176,C -2.0964,E1 24.8482,E2 288.7236} C_DIS
LIN {X -86.2512,Y 30.6435,Z 89,A 155.0964,B 24.9173,C -2.0996,E1 24.8494,E2 290.0284} C_DIS
LIN {X -85.4732,Y 32.751,Z 89,A 153.699,B 24.917,C -2.1042,E1 24.8508,E2 291.4228} C_DIS
LIN {X -84.6437,Y 34.8388,Z 89,A 152.2647,B 24.9167,C -2.1076,E1 24.8523,E2 292.8569} C_DIS
LIN {X -83.7633,Y 36.9055,Z 89,A 150.849,B 24.9164,C -2.1115,E1 24.8538,E2 294.271} C_DIS
LIN {X -82.8323,Y 38.9501,Z 89,A 149.4333,B 24.9161,C -2.1155,E1 24.8555,E2 295.6851} C_DIS
LIN {X -81.5179,Y 41.6295,Z 89,A 147.5233,B 24.9157,C -2.1197,E1 24.8579,E2 297.5952} C_DIS
LIN {X -80.1903,Y 44.1362,Z 89,A 145.7847,B 24.9152,C -2.126,E1 24.8602,E2 299.3281} C_DIS
LIN {X -79.083,Y 46.0909,Z 89,A 144.3695,B 24.9149,C -2.1298,E1 24.8621,E2 300.7417} C_DIS
LIN {X -78.0345,Y 47.8427,Z 89,A 143.0831,B 24.9147,C -2.1331,E1 24.864,E2 302.0266} C_DIS
LIN {X -76.8368,Y 49.7433,Z 89,A 141.6498,B 24.9144,C -2.1363,E1 24.8662,E2 303.4597} C_DIS
LIN {X -75.5929,Y 51.614,Z 89,A 140.2534,B 24.9141,C -2.1405,E1 24.8683,E2 304.8531} C_DIS
LIN {X -74.3035,Y 53.4536,Z 89,A 138.8387,B 24.9138,C -2.144,E1 24.8706,E2 306.2662} C_DIS
LIN {X -73.0236,Y 55.1888,Z 89,A 137.4772,B 24.9135,C -2.1473,E1 24.8729,E2 307.6264} C_DIS
LIN {X -71.4641,Y 57.1959,Z 89,A 135.8804,B 24.9132,C -2.1513,E1 24.8756,E2 309.2212} C_DIS
LIN {X -70.1699,Y 58.7749,Z 89,A 134.5804,B 24.913,C -2.154,E1 24.878,E2 310.5208} C_DIS
LIN {X -68.5715,Y 60.6336,Z 89,A 133.0522,B 24.9127,C -2.158,E1 24.8808,E2 312.0463} C_DIS
LIN {X -67.2014,Y 62.1472,Z 89,A 131.7485,B 24.9125,C -2.1604,E1 24.8832,E2 313.3499} C_DIS
LIN {X -65.5138,Y 63.9252,Z 89,A 130.0057,B 24.9127,C -2.1579,E1 24.8866,E2 315.1065} C_DIS
LIN {X -63.264,Y 66.1511,Z 89,A 128.2329,B 24.9118,C -2.1689,E1 24.8901,E2 316.8603} C_DIS
LIN {X -61.7213,Y 67.5922,Z 89,A 126.8581,B 24.9116,C -2.1703,E1 24.8929,E2 318.2373} C_DIS
LIN {X -59.9419,Y 69.1756,Z 89,A 125.406,B 24.9113,C -2.1749,E1 24.896,E2 319.6843} C_DIS
LIN {X -58.0686,Y 70.7568,Z 89,A 123.6584,B 24.9115,C -2.1717,E1 24.8998,E2 321.4461} C_DIS
LIN {X -55.4249,Y 72.8462,Z 89,A 121.745,B 24.9107,C -2.1822,E1 24.9039,E2 323.3416} C_DIS
LIN {X -53.2113,Y 74.4764,Z 89,A 119.8872,B 24.9107,C -2.1815,E1 24.9082,E2 325.2074} C_DIS
LIN {X -50.8536,Y 76.1078,Z 89,A 118.0157,B 24.9107,C -2.1826,E1 24.9125,E2 327.0826} C_DIS
LIN {X -48.0178,Y 77.928,Z 89,A 116.0955,B 24.9098,C -2.1924,E1 24.917,E2 328.9856} C_DIS
LIN {X -46.2674,Y 78.9787,Z 89,A 114.8126,B 24.9097,C -2.1946,E1 24.9201,E2 330.2673} C_DIS
LIN {X -44.1362,Y 80.1903,Z 89,A 113.2721,B 24.9095,C -2.197,E1 24.9238,E2 331.8063} C_DIS
LIN {X -41.1548,Y 81.7605,Z 89,A 111.1548,B 24.9092,C -2.2003,E1 24.9291,E2 333.9217} C_DIS
LIN {X -39.3206,Y 82.6571,Z 89,A 109.8541,B 24.9091,C -2.2016,E1 24.9323,E2 335.2227} C_DIS
LIN {X -37.2802,Y 83.5972,Z 89,A 108.4431,B 24.9089,C -2.2035,E1 24.9359,E2 336.6325} C_DIS
LIN {X -35.2174,Y 84.4869,Z 89,A 107.0325,B 24.9088,C -2.2054,E1 24.9395,E2 338.0419} C_DIS
LIN {X -33.1334,Y 85.3257,Z 89,A 105.6404,B 24.9086,C -2.2078,E1 24.9431,E2 339.4315} C_DIS
LIN {X -30.9717,Y 86.1342,Z 89,A 104.1822,B 24.9085,C -2.2092,E1 24.947,E2 340.8892} C_DIS
LIN {X -28.9068,Y 86.8487,Z 89,A 102.8019,B 24.9083,C -2.2104,E1 24.9506,E2 342.2691} C_DIS
LIN {X -25.9214,Y 87.7853,Z 89,A 100.7831,B 24.9083,C -2.2107,E1 24.956,E2 344.2907} C_DIS
LIN {X -23.3289,Y 88.5113,Z 89,A 99.1675,B 24.908,C -2.2147,E1 24.9604,E2 345.8994} C_DIS
LIN {X -21.3488,Y 89.0086,Z 89,A 97.8685,B 24.908,C -2.2152,E1 24.9639,E2 347.1989} C_DIS
LIN {X -19.158,Y 89.5057,Z 89,A 96.4598,B 24.9079,C -2.2164,E1 24.9677,E2 348.6067} C_DIS
LIN {X -16.7544,Y 89.9877,Z 89,A 94.9409,B 24.9077,C -2.2181,E1 24.9719,E2 350.1231} C_DIS
LIN {X -14.7431,Y 90.3379,Z 89,A 93.6425,B 24.9077,C -2.2184,E1 24.9754,E2 351.4221} C_DIS
LIN {X -12.5216,Y 90.6725,Z 89,A 92.234,B 24.9077,C -2.2192,E1 24.9793,E2 352.8297} C_DIS
LIN {X -10.2926,Y 90.9525,Z 89,A 90.8261,B 24.9076,C -2.22,E1 24.9832,E2 354.2369} C_DIS
LIN {X -8.0575,Y 91.1777,Z 89,A 89.4181,B 24.9076,C -2.2206,E1 24.9872,E2 355.644} C_DIS
LIN {X -5.8174,Y 91.348,Z 89,A 88.0107,B 24.9075,C -2.2211,E1 24.9911,E2 357.0507} C_DIS
LIN {X -3.3691,Y 91.4721,Z 89,A 86.2637,B 24.908,C -2.2147,E1 24.996,E2 358.8133} C_DIS
LIN {X -0.2049,Y 91.5328,Z 89,A 84.4931,B 24.9074,C -2.2221,E1 25.0009,E2 360.5665} C_DIS
LIN {X 2.7338,Y 91.4916,Z 89,A 82.5376,B 24.9077,C -2.2185,E1 25.0064,E2 362.5302} C_DIS
LIN {X 5.4057,Y 91.3733,Z 89,A 80.9778,B 24.9074,C -2.2223,E1 25.0107,E2 364.0803} C_DIS
LIN {X 7.8534,Y 91.1966,Z 89,A 79.4612,B 24.9074,C -2.2228,E1 25.0149,E2 365.5949} C_DIS
LIN {X 9.8853,Y 90.9977,Z 89,A 78.1647,B 24.9074,C -2.2221,E1 25.0185,E2 366.8924} C_DIS
LIN {X 12.8555,Y 90.6251,Z 89,A 76.2255,B 24.9076,C -2.2195,E1 25.0239,E2 368.8361} C_DIS
LIN {X 15.6488,Y 90.1865,Z 89,A 74.5415,B 24.9074,C -2.2217,E1 25.0285,E2 370.5131} C_DIS
LIN {X 17.6562,Y 89.814,Z 89,A 73.2645,B 24.9074,C -2.2213,E1 25.032,E2 371.7897} C_DIS
LIN {X 20.0552,Y 89.31,Z 89,A 71.7319,B 24.9075,C -2.2206,E1 25.0362,E2 373.322} C_DIS
LIN {X 22.0448,Y 88.8388,Z 89,A 70.4539,B 24.9075,C -2.2199,E1 25.0397,E2 374.5997} C_DIS
LIN {X 24.4133,Y 88.2184,Z 89,A 68.9228,B 24.9076,C -2.219,E1 25.0438,E2 376.1306} C_DIS
LIN {X 26.3745,Y 87.6509,Z 89,A 67.6286,B 24.9078,C -2.2175,E1 25.0473,E2 377.426} C_DIS
LIN {X 29.1486,Y 86.7672,Z 89,A 65.7499,B 24.908,C -2.2142,E1 25.0523,E2 379.3091} C_DIS
LIN {X 31.6997,Y 85.8687,Z 89,A 64.1194,B 24.908,C -2.2148,E1 25.0565,E2 380.9349} C_DIS
LIN {X 33.7974,Y 85.0649,Z 89,A 62.7164,B 24.908,C -2.2135,E1 25.0602,E2 382.3378} C_DIS
LIN {X 35.8748,Y 84.2098,Z 89,A 61.3319,B 24.9082,C -2.2128,E1 25.0637,E2 383.7208} C_DIS
LIN {X 38.1175,Y 83.2199,Z 89,A 59.8009,B 24.9082,C -2.2111,E1 25.0676,E2 385.2518} C_DIS
LIN {X 39.9636,Y 82.3481,Z 89,A 58.5266,B 24.9084,C -2.2097,E1 25.0709,E2 386.5262} C_DIS
LIN {X 41.9014,Y 81.3789,Z 89,A 57.1405,B 24.9086,C -2.207,E1 25.0743,E2 387.9149} C_DIS
LIN {X 44.5696,Y 79.9483,Z 89,A 55.1545,B 24.9091,C -2.2013,E1 25.0792,E2 389.9087} C_DIS
LIN {X 47.0579,Y 78.5114,Z 89,A 53.3213,B 24.9094,C -2.1974,E1 25.0836,E2 391.7454} C_DIS
LIN {X 49.7434,Y 76.8368,Z 89,A 51.4988,B 24.9092,C -2.1999,E1 25.0879,E2 393.5563} C_DIS
LIN {X 52.2049,Y 75.1853,Z 89,A 49.5745,B 24.9097,C -2.1945,E1 25.0923,E2 395.4868} C_DIS
LIN {X 54.3614,Y 73.6419,Z 89,A 47.9959,B 24.9097,C -2.1945,E1 25.0959,E2 397.0599} C_DIS
LIN {X 56.1523,Y 72.2857,Z 89,A 46.6136,B 24.9098,C -2.1927,E1 25.099,E2 398.4412} C_DIS
LIN {X 58.0686,Y 70.7568,Z 89,A 45.0854,B 24.91,C -2.1901,E1 25.1023,E2 399.9699} C_DIS
LIN {X 60.147,Y 68.9965,Z 89,A 43.2823,B 24.9106,C -2.1834,E1 25.1061,E2 401.7817} C_DIS
LIN {X 62.2006,Y 67.1524,Z 89,A 41.6594,B 24.9106,C -2.1836,E1 25.1095,E2 403.3977} C_DIS
LIN {X 63.9252,Y 65.5138,Z 89,A 40.185,B 24.9108,C -2.181,E1 25.1124,E2 404.8721} C_DIS
LIN {X 65.3697,Y 64.071,Z 89,A 38.9262,B 24.9109,C -2.179,E1 25.1149,E2 406.1303} C_DIS
LIN {X 66.9224,Y 62.4475,Z 89,A 37.4952,B 24.9113,C -2.175,E1 25.1176,E2 407.5644} C_DIS
Enddeposition()
END
